KUKA KRL program: MyProgram_159().src

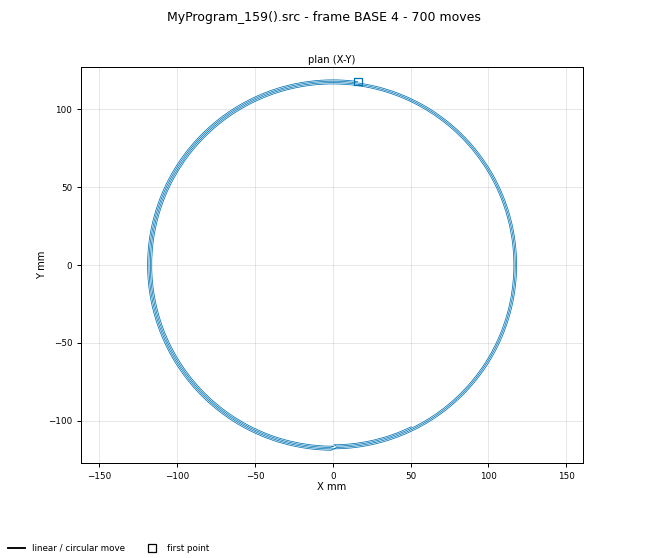
[picture p0: tool path of MyProgram_159().src in frame BASE 4, 700 of 700 moves have a stored position in this frame; points joined in program order, loops and branches not executed]
&ACCESS RVP
&REL 1
&PARAM TEMPLATE = C:\KRC\Roboter\Template\vorgabe
&PARAM EDITMASK = *
DEF MyProgram_159()
; ---- Setting reference (Base) ----
$BASE = BASE_DATA[4]

; --------------------------
; ---- Setting tool (TCP) ----
$TOOL = TOOL_DATA[3]
; --------------------------

$VEL.CP = VEL_APROX_PRINT
Startdeposition()
$VEL.CP = VEL_PRINT
LIN {X 16.0086,Y 117.8693,Z 122,A 78.2901,B 24.9375,C -1.8274,E1 25.0208,E2 367.7031} C_DIS
LIN {X 13.1111,Y 118.2266,Z 122,A 79.7079,B 24.9374,C -1.8281,E1 25.0168,E2 366.2845} C_DIS
LIN {X 10.2057,Y 118.5128,Z 122,A 81.1015,B 24.9374,C -1.8277,E1 25.013,E2 364.8927} C_DIS
LIN {X 6.984,Y 118.7447,Z 122,A 82.7398,B 24.9371,C -1.8315,E1 25.0084,E2 363.2462} C_DIS
LIN {X 2.9192,Y 118.9156,Z 122,A 84.6175,B 24.9374,C -1.8276,E1 25.0032,E2 361.3781} C_DIS
LIN {X 0,Y 118.9514,Z 122,A 86.0242,B 24.9374,C -1.8274,E1 24.9992,E2 359.9721} C_DIS
LIN {X -3.3524,Y 118.9023,Z 122,A 87.6856,B 24.9373,C -1.8291,E1 24.9946,E2 358.3065} C_DIS
LIN {X -7.2942,Y 118.7275,Z 122,A 89.5422,B 24.9375,C -1.8264,E1 24.9894,E2 356.4558} C_DIS
LIN {X -10.2057,Y 118.5128,Z 122,A 90.9498,B 24.9375,C -1.8258,E1 24.9855,E2 355.0489} C_DIS
LIN {X -13.2482,Y 118.2106,Z 122,A 92.3641,B 24.9377,C -1.8224,E1 24.9816,E2 353.6418} C_DIS
LIN {X -16.0086,Y 117.8693,Z 122,A 93.766,B 24.9377,C -1.8244,E1 24.9777,E2 352.2344} C_DIS
LIN {X -19.1267,Y 117.4024,Z 122,A 95.1851,B 24.938,C -1.8189,E1 24.9738,E2 350.8269} C_DIS
LIN {X -22.2224,Y 116.8552,Z 122,A 96.604,B 24.9384,C -1.8135,E1 24.9699,E2 349.4193} C_DIS
LIN {X -24.7181,Y 116.3543,Z 122,A 97.9954,B 24.9379,C -1.8198,E1 24.9661,E2 348.0115} C_DIS
LIN {X -27.4847,Y 115.7326,Z 122,A 99.4967,B 24.9376,C -1.8245,E1 24.962,E2 346.497} C_DIS
LIN {X -31.7259,Y 114.6425,Z 122,A 101.5145,B 24.938,C -1.8183,E1 24.9566,E2 344.491} C_DIS
LIN {X -34.5298,Y 113.8294,Z 122,A 102.9241,B 24.9381,C -1.8169,E1 24.9528,E2 343.0823} C_DIS
LIN {X -37.3129,Y 112.9477,Z 122,A 104.3341,B 24.9382,C -1.8154,E1 24.949,E2 341.6734} C_DIS
LIN {X -40.0735,Y 111.998,Z 122,A 105.7441,B 24.9383,C -1.8137,E1 24.9453,E2 340.2645} C_DIS
LIN {X -42.81,Y 110.9808,Z 122,A 107.1543,B 24.9385,C -1.812,E1 24.9417,E2 338.8553} C_DIS
LIN {X -45.5207,Y 109.8968,Z 122,A 108.5648,B 24.9385,C -1.8102,E1 24.938,E2 337.4459} C_DIS
LIN {X -48.204,Y 108.7465,Z 122,A 110.0438,B 24.9385,C -1.8113,E1 24.9342,E2 335.9608} C_DIS
LIN {X -50.8583,Y 107.5308,Z 122,A 111.3866,B 24.9388,C -1.8064,E1 24.9308,E2 334.6265} C_DIS
LIN {X -53.4819,Y 106.2503,Z 122,A 112.7979,B 24.939,C -1.8043,E1 24.9273,E2 333.2164} C_DIS
LIN {X -56.3435,Y 104.7592,Z 122,A 114.2234,B 24.9395,C -1.7961,E1 24.9238,E2 331.8064} C_DIS
LIN {X -58.6309,Y 103.4981,Z 122,A 115.6207,B 24.9393,C -1.7999,E1 24.9204,E2 330.396} C_DIS
LIN {X -61.1532,Y 102.028,Z 122,A 117.0324,B 24.9394,C -1.7976,E1 24.917,E2 328.9856} C_DIS
LIN {X -63.6387,Y 100.4965,Z 122,A 118.4444,B 24.9396,C -1.7952,E1 24.9137,E2 327.5749} C_DIS
LIN {X -66.0859,Y 98.9045,Z 122,A 119.8565,B 24.9398,C -1.7927,E1 24.9104,E2 326.1641} C_DIS
LIN {X -68.6207,Y 97.1619,Z 122,A 121.276,B 24.9401,C -1.787,E1 24.9071,E2 324.7532} C_DIS
LIN {X -70.8593,Y 95.5427,Z 122,A 122.6815,B 24.9401,C -1.7874,E1 24.9039,E2 323.3417} C_DIS
LIN {X -73.1827,Y 93.7749,Z 122,A 124.1704,B 24.9401,C -1.788,E1 24.9006,E2 321.8462} C_DIS
LIN {X -75.9227,Y 91.5678,Z 122,A 125.7971,B 24.9405,C -1.7813,E1 24.8971,E2 320.2291} C_DIS
LIN {X -78.7953,Y 89.1108,Z 122,A 127.6267,B 24.9408,C -1.7775,E1 24.8933,E2 318.4014} C_DIS
LIN {X -80.9584,Y 87.1502,Z 122,A 129.0403,B 24.941,C -1.7745,E1 24.8904,E2 316.9892} C_DIS
LIN {X -83.0728,Y 85.1372,Z 122,A 130.4536,B 24.9412,C -1.7715,E1 24.8875,E2 315.5773} C_DIS
LIN {X -85.1372,Y 83.0728,Z 122,A 131.8674,B 24.9414,C -1.7683,E1 24.8848,E2 314.165} C_DIS
LIN {X -87.2091,Y 80.8943,Z 122,A 133.2852,B 24.9417,C -1.7634,E1 24.8821,E2 312.7527} C_DIS
LIN {X -89.1108,Y 78.7953,Z 122,A 134.6952,B 24.9418,C -1.7618,E1 24.8794,E2 311.3402} C_DIS
LIN {X -91.2779,Y 76.2716,Z 122,A 136.1286,B 24.9426,C -1.7505,E1 24.8769,E2 309.9272} C_DIS
LIN {X -92.8698,Y 74.3279,Z 122,A 137.5238,B 24.9423,C -1.7551,E1 24.8744,E2 308.5145} C_DIS
LIN {X -94.6659,Y 72.0264,Z 122,A 138.9381,B 24.9425,C -1.7517,E1 24.872,E2 307.1016} C_DIS
LIN {X -96.405,Y 69.6815,Z 122,A 140.3529,B 24.9427,C -1.7482,E1 24.8697,E2 305.6883} C_DIS
LIN {X -98.0861,Y 67.2946,Z 122,A 141.7675,B 24.943,C -1.7446,E1 24.8674,E2 304.2753} C_DIS
LIN {X -99.708,Y 64.8672,Z 122,A 143.25,B 24.943,C -1.7438,E1 24.8651,E2 302.7872} C_DIS
LIN {X -101.2699,Y 62.4007,Z 122,A 144.5972,B 24.9434,C -1.7373,E1 24.8632,E2 301.4486} C_DIS
LIN {X -102.7708,Y 59.8966,Z 122,A 146.0608,B 24.9435,C -1.7356,E1 24.8611,E2 299.9814} C_DIS
LIN {X -104.2098,Y 57.3564,Z 122,A 147.4273,B 24.9439,C -1.7298,E1 24.8592,E2 298.6216} C_DIS
LIN {X -105.586,Y 54.7817,Z 122,A 148.8428,B 24.9442,C -1.726,E1 24.8574,E2 297.2076} C_DIS
LIN {X -106.8986,Y 52.174,Z 122,A 150.258,B 24.9444,C -1.7222,E1 24.8556,E2 295.794} C_DIS
LIN {X -108.1468,Y 49.5349,Z 122,A 151.6736,B 24.9447,C -1.7183,E1 24.854,E2 294.3799} C_DIS
LIN {X -109.3299,Y 46.8659,Z 122,A 153.0891,B 24.9449,C -1.7144,E1 24.8524,E2 292.9659} C_DIS
LIN {X -110.4471,Y 44.1687,Z 122,A 154.5047,B 24.9452,C -1.7104,E1 24.8509,E2 291.5519} C_DIS
LIN {X -111.4978,Y 41.4449,Z 122,A 155.9204,B 24.9454,C -1.7064,E1 24.8495,E2 290.1377} C_DIS
LIN {X -112.4813,Y 38.6961,Z 122,A 157.4741,B 24.9454,C -1.7082,E1 24.8481,E2 288.5709} C_DIS
LIN {X -113.588,Y 35.3084,Z 122,A 158.9656,B 24.9463,C -1.6934,E1 24.8468,E2 287.1063} C_DIS
LIN {X -114.4079,Y 32.5539,Z 122,A 160.4567,B 24.9463,C -1.6934,E1 24.8457,E2 285.6064} C_DIS
LIN {X -115.1723,Y 29.7364,Z 122,A 161.8742,B 24.9465,C -1.6894,E1 24.8446,E2 284.1903} C_DIS
LIN {X -116.0611,Y 26.0624,Z 122,A 163.7079,B 24.9469,C -1.6841,E1 24.8435,E2 282.3586} C_DIS
LIN {X -116.6658,Y 23.2063,Z 122,A 165.2237,B 24.9469,C -1.6841,E1 24.8426,E2 280.8337} C_DIS
LIN {X -117.4409,Y 18.8964,Z 122,A 167.248,B 24.9475,C -1.6737,E1 24.8417,E2 278.8222} C_DIS
LIN {X -117.8693,Y 16.0086,Z 122,A 168.6643,B 24.9478,C -1.6696,E1 24.8411,E2 277.4074} C_DIS
LIN {X -118.2266,Y 13.1111,Z 122,A 170.2103,B 24.9477,C -1.6708,E1 24.8406,E2 275.849} C_DIS
LIN {X -118.5128,Y 10.2057,Z 122,A 171.4964,B 24.9483,C -1.6612,E1 24.8403,E2 274.5782} C_DIS
LIN {X -118.7486,Y 6.9139,Z 122,A 172.9304,B 24.949,C -1.6495,E1 24.84,E2 273.1635} C_DIS
LIN {X -118.8708,Y 4.3783,Z 122,A 174.3286,B 24.9488,C -1.6529,E1 24.8399,E2 271.7489} C_DIS
LIN {X -118.9424,Y 1.4597,Z 122,A 175.741,B 24.9491,C -1.6485,E1 24.8398,E2 270.3382} C_DIS
LIN {X -118.9424,Y -1.4597,Z 122,A 177.3307,B 24.9489,C -1.6517,E1 24.8398,E2 268.7315} C_DIS
LIN {X -118.8081,Y -5.8367,Z 122,A 179.285,B 24.9497,C -1.6383,E1 24.84,E2 266.7973} C_DIS
LIN {X -118.6291,Y -8.7506,Z 122,A -179.2988,B 24.95,C -1.6342,E1 24.8403,E2 265.3825} C_DIS
LIN {X -118.3786,Y -11.6593,Z 122,A -177.7646,B 24.95,C -1.635,E1 24.8407,E2 263.837} C_DIS
LIN {X -118.0568,Y -14.5609,Z 122,A -176.2909,B 24.95,C -1.6334,E1 24.8412,E2 262.3584} C_DIS
LIN {X -117.6639,Y -17.4538,Z 122,A -175.0509,B 24.9507,C -1.6218,E1 24.8417,E2 261.1385} C_DIS
LIN {X -117.2002,Y -20.3362,Z 122,A -173.6352,B 24.951,C -1.6178,E1 24.8423,E2 259.724} C_DIS
LIN {X -116.6658,Y -23.2063,Z 122,A -172.2193,B 24.9512,C -1.6137,E1 24.8431,E2 258.3094} C_DIS
LIN {X -116.0611,Y -26.0624,Z 122,A -170.8033,B 24.9514,C -1.6097,E1 24.8439,E2 256.8947} C_DIS
LIN {X -115.3866,Y -28.9028,Z 122,A -169.3877,B 24.9517,C -1.6058,E1 24.8449,E2 255.4803} C_DIS
LIN {X -114.4951,Y -32.2459,Z 122,A -167.9472,B 24.9526,C -1.5911,E1 24.8459,E2 254.0663} C_DIS
LIN {X -113.8294,Y -34.5298,Z 122,A -166.5567,B 24.9522,C -1.5979,E1 24.847,E2 252.6516} C_DIS
LIN {X -112.9477,Y -37.3129,Z 122,A -165.1412,B 24.9524,C -1.594,E1 24.8482,E2 251.2372} C_DIS
LIN {X -111.9561,Y -40.1883,Z 122,A -163.7202,B 24.9528,C -1.5878,E1 24.8495,E2 249.8231} C_DIS
LIN {X -110.9808,Y -42.81,Z 122,A -162.3107,B 24.9528,C -1.5864,E1 24.8509,E2 248.4089} C_DIS
LIN {X -109.8968,Y -45.5207,Z 122,A -160.8955,B 24.9531,C -1.5826,E1 24.8524,E2 246.9948} C_DIS
LIN {X -108.7465,Y -48.204,Z 122,A -159.4806,B 24.9533,C -1.5789,E1 24.854,E2 245.5808} C_DIS
LIN {X -107.5308,Y -50.8583,Z 122,A -158.0655,B 24.9535,C -1.5753,E1 24.8557,E2 244.1668} C_DIS
LIN {X -106.0721,Y -53.8304,Z 122,A -156.6322,B 24.9542,C -1.5639,E1 24.8574,E2 242.7527} C_DIS
LIN {X -104.9058,Y -56.0733,Z 122,A -155.236,B 24.9539,C -1.5681,E1 24.8593,E2 241.3392} C_DIS
LIN {X -103.4981,Y -58.6309,Z 122,A -153.8215,B 24.9541,C -1.5646,E1 24.8612,E2 239.9255} C_DIS
LIN {X -102.028,Y -61.1532,Z 122,A -152.4071,B 24.9543,C -1.5612,E1 24.8632,E2 238.5121} C_DIS
LIN {X -100.4965,Y -63.6387,Z 122,A -150.9929,B 24.9545,C -1.5578,E1 24.8653,E2 237.0987} C_DIS
LIN {X -98.9045,Y -66.0859,Z 122,A -149.5789,B 24.9547,C -1.5545,E1 24.8675,E2 235.6854} C_DIS
LIN {X -97.2529,Y -68.4932,Z 122,A -148.1649,B 24.9549,C -1.5513,E1 24.8697,E2 234.2722} C_DIS
LIN {X -95.5427,Y -70.8593,Z 122,A -146.7512,B 24.9551,C -1.5481,E1 24.8721,E2 232.8592} C_DIS
LIN {X -93.7749,Y -73.1827,Z 122,A -145.3375,B 24.9553,C -1.545,E1 24.8745,E2 231.4463} C_DIS
LIN {X -91.9507,Y -75.462,Z 122,A -143.9239,B 24.9555,C -1.5419,E1 24.877,E2 230.0333} C_DIS
LIN {X -90.0711,Y -77.6958,Z 122,A -142.5105,B 24.9556,C -1.5389,E1 24.8795,E2 228.6206} C_DIS
LIN {X -88.1372,Y -79.8829,Z 122,A -141.0974,B 24.9558,C -1.536,E1 24.8822,E2 227.2081} C_DIS
LIN {X -86.1502,Y -82.0218,Z 122,A -139.6846,B 24.956,C -1.5332,E1 24.8849,E2 225.7959} C_DIS
LIN {X -84.1113,Y -84.1113,Z 122,A -138.2717,B 24.9561,C -1.5305,E1 24.8876,E2 224.3834} C_DIS
LIN {X -82.0218,Y -86.1502,Z 122,A -136.8593,B 24.9563,C -1.5278,E1 24.8905,E2 222.9716} C_DIS
LIN {X -79.8829,Y -88.1372,Z 122,A -135.4465,B 24.9564,C -1.5252,E1 24.8934,E2 221.5593} C_DIS
LIN {X -77.6958,Y -90.0711,Z 122,A -134.0346,B 24.9566,C -1.5227,E1 24.8963,E2 220.1478} C_DIS
LIN {X -75.462,Y -91.9507,Z 122,A -132.6226,B 24.9567,C -1.5202,E1 24.8994,E2 218.7362} C_DIS
LIN {X -72.8436,Y -94.0362,Z 122,A -131.1909,B 24.9573,C -1.5094,E1 24.9025,E2 217.325} C_DIS
LIN {X -70.8593,Y -95.5427,Z 122,A -129.7991,B 24.957,C -1.5156,E1 24.9056,E2 215.9134} C_DIS
LIN {X -68.4932,Y -97.2529,Z 122,A -128.3878,B 24.957,C -1.5135,E1 24.9088,E2 214.5024} C_DIS
LIN {X -66.0859,Y -98.9045,Z 122,A -126.9767,B 24.9572,C -1.5114,E1 24.9121,E2 213.0914} C_DIS
LIN {X -63.6387,Y -100.4965,Z 122,A -125.5655,B 24.9573,C -1.5094,E1 24.9154,E2 211.6805} C_DIS
LIN {X -61.1532,Y -102.028,Z 122,A -124.1547,B 24.9574,C -1.5075,E1 24.9188,E2 210.2699} C_DIS
LIN {X -58.6309,Y -103.4981,Z 122,A -122.7442,B 24.9575,C -1.5057,E1 24.9222,E2 208.8595} C_DIS
LIN {X -56.0733,Y -104.9058,Z 122,A -121.3338,B 24.9576,C -1.5039,E1 24.9257,E2 207.4491} C_DIS
LIN {X -53.4819,Y -106.2503,Z 122,A -119.886,B 24.9576,C -1.504,E1 24.9293,E2 205.9973} C_DIS
LIN {X -50.8583,Y -107.5308,Z 122,A -118.5141,B 24.9578,C -1.5008,E1 24.9327,E2 204.6295} C_DIS
LIN {X -48.204,Y -108.7465,Z 122,A -117.1043,B 24.9578,C -1.4994,E1 24.9363,E2 203.2197} C_DIS
LIN {X -45.5207,Y -109.8968,Z 122,A -115.695,B 24.958,C -1.498,E1 24.9399,E2 201.8104} C_DIS
LIN {X -42.81,Y -110.9808,Z 122,A -114.119,B 24.9576,C -1.5043,E1 24.9441,E2 200.2161} C_DIS
LIN {X -39.8038,Y -112.0926,Z 122,A -112.8631,B 24.9584,C -1.49,E1 24.9473,E2 198.9917} C_DIS
LIN {X -37.3129,Y -112.9477,Z 122,A -111.4682,B 24.9582,C -1.4946,E1 24.951,E2 197.5832} C_DIS
LIN {X -34.5298,Y -113.8294,Z 122,A -110.0595,B 24.9582,C -1.4936,E1 24.9548,E2 196.1743} C_DIS
LIN {X -31.6187,Y -114.6714,Z 122,A -108.6462,B 24.9584,C -1.4906,E1 24.9586,E2 194.7659} C_DIS
LIN {X -28.9028,Y -115.3866,Z 122,A -107.2432,B 24.9583,C -1.4921,E1 24.9624,E2 193.3575} C_DIS
LIN {X -26.0624,Y -116.0611,Z 122,A -105.8354,B 24.9583,C -1.4914,E1 24.9662,E2 191.9494} C_DIS
LIN {X -23.2063,Y -116.6658,Z 122,A -104.3529,B 24.9582,C -1.4943,E1 24.9703,E2 190.4583} C_DIS
LIN {X -19.7453,Y -117.2989,Z 122,A -102.732,B 24.9584,C -1.4904,E1 24.9747,E2 188.8451} C_DIS
LIN {X -16.0086,Y -117.8693,Z 122,A -100.8392,B 24.9582,C -1.4932,E1 24.98,E2 186.944} C_DIS
LIN {X -13.1111,Y -118.2266,Z 122,A -99.5036,B 24.9584,C -1.4898,E1 24.9837,E2 185.6156} C_DIS
LIN {X -10.2057,Y -118.5128,Z 122,A -98.0971,B 24.9584,C -1.4897,E1 24.9876,E2 184.2086} C_DIS
LIN {X -7.2942,Y -118.7275,Z 122,A -96.6908,B 24.9584,C -1.4897,E1 24.9915,E2 182.8017} C_DIS
LIN {X -4.3783,Y -118.8708,Z 122,A -95.2849,B 24.9584,C -1.4898,E1 24.9954,E2 181.3953} C_DIS
LIN {X -1.1166,Y -118.9445,Z 122,A -93.6416,B 24.9582,C -1.4934,E1 25,E2 179.7433} C_DIS
LIN {X -1.1166,Y -118.9445,Z 122,A -93.6416,B 24.9582,C -1.4934,E1 25,E2 179.7433} C_DIS
Enddeposition()
LIN {X 0.837,Y -118.0667,Z 122,A -93.3866,B 24.9591,C -1.4776,E1 25.0006,E2 179.5259} C_DIS
Startdeposition()
$VEL.CP = VEL_PRINT
LIN {X -2.5203,Y -118.0457,Z 122,A -95.0963,B 24.9593,C -1.4736,E1 24.9958,E2 181.2451} C_DIS
LIN {X -6.0284,Y -117.9191,Z 122,A -96.9279,B 24.9596,C -1.4677,E1 24.9907,E2 183.0911} C_DIS
LIN {X -9.7991,Y -117.6654,Z 122,A -98.7213,B 24.9596,C -1.4695,E1 24.9857,E2 184.8809} C_DIS
LIN {X -13.6232,Y -117.2835,Z 122,A -100.5453,B 24.9594,C -1.4716,E1 24.9806,E2 186.701} C_DIS
LIN {X -17.1647,Y -116.8191,Z 122,A -102.3364,B 24.9596,C -1.4694,E1 24.9757,E2 188.4989} C_DIS
LIN {X -20.8111,Y -116.2235,Z 122,A -104.0964,B 24.9594,C -1.4714,E1 24.9708,E2 190.2557} C_DIS
LIN {X -24.1501,Y -115.5766,Z 122,A -105.8865,B 24.9597,C -1.4659,E1 24.9659,E2 192.0609} C_DIS
LIN {X -28.319,Y -114.6262,Z 122,A -107.7431,B 24.9591,C -1.4767,E1 24.9609,E2 193.8945} C_DIS
LIN {X -31.6333,Y -113.7571,Z 122,A -109.4534,B 24.9592,C -1.4756,E1 24.9563,E2 195.61} C_DIS
LIN {X -35.4313,Y -112.6316,Z 122,A -111.4026,B 24.9592,C -1.4758,E1 24.9511,E2 197.562} C_DIS
LIN {X -39.6049,Y -111.2329,Z 122,A -113.4657,B 24.9589,C -1.4808,E1 24.9456,E2 199.6172} C_DIS
LIN {X -43.033,Y -109.9508,Z 122,A -115.3202,B 24.959,C -1.4791,E1 24.9408,E2 201.4797} C_DIS
LIN {X -46.5467,Y -108.5122,Z 122,A -117.2594,B 24.9591,C -1.4768,E1 24.9358,E2 203.4289} C_DIS
LIN {X -49.8822,Y -107.0176,Z 122,A -118.9207,B 24.9588,C -1.4837,E1 24.9316,E2 205.0777} C_DIS
LIN {X -52.9112,Y -105.5542,Z 122,A -120.5495,B 24.9586,C -1.4859,E1 24.9275,E2 206.7057} C_DIS
LIN {X -56.2696,Y -103.8014,Z 122,A -122.3858,B 24.9585,C -1.4884,E1 24.923,E2 208.541} C_DIS
LIN {X -59.4142,Y -102.0362,Z 122,A -125.1607,B 24.9608,C -1.4469,E1 24.9161,E2 211.4229} C_DIS
LIN {X -64.7113,Y -98.7602,Z 122,A -127.2367,B 24.9583,C -1.4921,E1 24.9114,E2 213.3982} C_DIS
LIN {X -67.4344,Y -96.9207,Z 122,A -128.7977,B 24.9581,C -1.4962,E1 24.9078,E2 214.9547} C_DIS
LIN {X -70.4261,Y -94.771,Z 122,A -130.6293,B 24.958,C -1.4974,E1 24.9037,E2 216.7899} C_DIS
LIN {X -73.6051,Y -92.3231,Z 122,A -133.3064,B 24.9595,C -1.47,E1 24.8977,E2 219.5422} C_DIS
LIN {X -77.5667,Y -89.0192,Z 122,A -134.7328,B 24.9567,C -1.5206,E1 24.8949,E2 220.8536} C_DIS
LIN {X -80.6537,Y -86.2328,Z 122,A -137.0863,B 24.9573,C -1.5103,E1 24.8899,E2 223.241} C_DIS
LIN {X -82.9849,Y -83.9912,Z 122,A -138.6859,B 24.9571,C -1.5124,E1 24.8867,E2 224.8424} C_DIS
LIN {X -85.3632,Y -81.5744,Z 122,A -140.3333,B 24.9569,C -1.5159,E1 24.8835,E2 226.4886} C_DIS
LIN {X -87.9813,Y -78.742,Z 122,A -142.2473,B 24.9569,C -1.5183,E1 24.8799,E2 228.4053} C_DIS
LIN {X -90.2888,Y -76.0878,Z 122,A -143.9596,B 24.9566,C -1.522,E1 24.8768,E2 230.1165} C_DIS
LIN {X -92.7396,Y -73.078,Z 122,A -145.7909,B 24.9562,C -1.5288,E1 24.8736,E2 231.9403} C_DIS
LIN {X -95.2869,Y -69.7238,Z 122,A -147.8273,B 24.9559,C -1.5342,E1 24.8702,E2 233.9737} C_DIS
LIN {X -97.3807,Y -66.7718,Z 122,A -149.545,B 24.9556,C -1.5402,E1 24.8675,E2 235.6854} C_DIS
LIN {X -99.1458,Y -64.1192,Z 122,A -151.191,B 24.9556,C -1.5401,E1 24.8649,E2 237.34} C_DIS
LIN {X -101.046,Y -61.0803,Z 122,A -152.8963,B 24.9552,C -1.5461,E1 24.8625,E2 239.0397} C_DIS
LIN {X -102.7863,Y -58.1065,Z 122,A -154.6916,B 24.9552,C -1.5455,E1 24.8599,E2 240.8458} C_DIS
LIN {X -104.6351,Y -54.7049,Z 122,A -156.4189,B 24.9546,C -1.557,E1 24.8577,E2 242.5548} C_DIS
LIN {X -106.1616,Y -51.6825,Z 122,A -158.3147,B 24.9549,C -1.5511,E1 24.8553,E2 244.4749} C_DIS
LIN {X -108.0733,Y -47.5535,Z 122,A -160.645,B 24.9549,C -1.5524,E1 24.8526,E2 246.8149} C_DIS
LIN {X -109.8468,Y -43.298,Z 122,A -162.6472,B 24.9539,C -1.5687,E1 24.8506,E2 248.7893} C_DIS
LIN {X -111.1689,Y -39.7858,Z 122,A -164.3767,B 24.9533,C -1.5779,E1 24.8489,E2 250.5067} C_DIS
LIN {X -112.2303,Y -36.681,Z 122,A -166.101,B 24.9533,C -1.5773,E1 24.8474,E2 252.2424} C_DIS
LIN {X -113.1981,Y -33.5739,Z 122,A -167.6026,B 24.9529,C -1.5853,E1 24.8462,E2 253.7335} C_DIS
LIN {X -114.0754,Y -30.4619,Z 122,A -169.6456,B 24.9538,C -1.5707,E1 24.8446,E2 255.8233} C_DIS
LIN {X -114.957,Y -26.9451,Z 122,A -170.7843,B 24.9519,C -1.6017,E1 24.8439,E2 256.8947} C_DIS
LIN {X -115.6853,Y -23.6207,Z 122,A -172.8482,B 24.9526,C -1.5899,E1 24.8427,E2 258.9989} C_DIS
LIN {X -116.6652,Y -18.173,Z 122,A -175.4722,B 24.952,C -1.601,E1 24.8415,E2 261.6121} C_DIS
LIN {X -117.2671,Y -13.7637,Z 122,A -177.5041,B 24.9512,C -1.6131,E1 24.8408,E2 263.6272} C_DIS
LIN {X -117.5907,Y -10.6525,Z 122,A -179.1069,B 24.9512,C -1.6145,E1 24.8403,E2 265.2362} C_DIS
LIN {X -117.8809,Y -6.7187,Z 122,A 178.9732,B 24.9508,C -1.6205,E1 24.84,E2 267.1535} C_DIS
LIN {X -118.0266,Y -3.2916,Z 122,A 177.31,B 24.9505,C -1.6259,E1 24.8398,E2 268.8137} C_DIS
LIN {X -118.0707,Y 0.6735,Z 122,A 175.2326,B 24.9505,C -1.6259,E1 24.8398,E2 270.9036} C_DIS
LIN {X -117.999,Y 4.191,Z 122,A 173.6973,B 24.9497,C -1.6385,E1 24.8399,E2 272.4182} C_DIS
LIN {X -117.8225,Y 7.6782,Z 122,A 172.1845,B 24.9489,C -1.6515,E1 24.8402,E2 273.9091} C_DIS
LIN {X -117.6304,Y 10.2227,Z 122,A 170.5906,B 24.9495,C -1.6409,E1 24.8405,E2 275.5378} C_DIS
LIN {X -117.2382,Y 14.0105,Z 122,A 168.906,B 24.9488,C -1.6537,E1 24.841,E2 277.2021} C_DIS
LIN {X -116.7982,Y 17.3099,Z 122,A 167.3023,B 24.9484,C -1.6594,E1 24.8417,E2 278.8018} C_DIS
LIN {X -116.0604,Y 21.7112,Z 122,A 163.9484,B 24.9509,C -1.6182,E1 24.8434,E2 282.2738} C_DIS
LIN {X -114.6541,Y 28.2045,Z 122,A 161.7774,B 24.9477,C -1.6712,E1 24.8447,E2 284.331} C_DIS
LIN {X -113.6608,Y 31.9732,Z 122,A 159.8393,B 24.9474,C -1.6753,E1 24.8462,E2 286.2706} C_DIS
LIN {X -112.4649,Y 35.9559,Z 122,A 157.7732,B 24.9471,C -1.6798,E1 24.8479,E2 288.3379} C_DIS
LIN {X -111.1922,Y 39.7203,Z 122,A 155.8664,B 24.9467,C -1.6867,E1 24.8496,E2 290.2391} C_DIS
LIN {X -109.9722,Y 42.9785,Z 122,A 154.2022,B 24.9463,C -1.693,E1 24.8513,E2 291.8977} C_DIS
LIN {X -108.4935,Y 46.5895,Z 122,A 152.254,B 24.9461,C -1.6965,E1 24.8534,E2 293.8483} C_DIS
LIN {X -106.9839,Y 49.9548,Z 122,A 150.543,B 24.9455,C -1.7052,E1 24.8553,E2 295.5479} C_DIS
LIN {X -105.5465,Y 52.9268,Z 122,A 148.9998,B 24.945,C -1.7125,E1 24.8572,E2 297.0821} C_DIS
LIN {X -104.1322,Y 55.6598,Z 122,A 147.2749,B 24.9454,C -1.7074,E1 24.8595,E2 298.8284} C_DIS
LIN {X -101.2999,Y 60.6614,Z 122,A 144.5478,B 24.9447,C -1.7181,E1 24.8633,E2 301.5441} C_DIS
LIN {X -99.4431,Y 63.6562,Z 122,A 142.8906,B 24.9442,C -1.7252,E1 24.8657,E2 303.1929} C_DIS
LIN {X -97.7178,Y 66.274,Z 122,A 141.3586,B 24.944,C -1.729,E1 24.8681,E2 304.7233} C_DIS
LIN {X -94.6762,Y 70.5522,Z 122,A 138.6995,B 24.9438,C -1.7314,E1 24.8725,E2 307.3897} C_DIS
LIN {X -92.2919,Y 73.6445,Z 122,A 136.8665,B 24.9433,C -1.739,E1 24.8756,E2 309.2131} C_DIS
LIN {X -89.7223,Y 76.7526,Z 122,A 134.9443,B 24.9429,C -1.7456,E1 24.8791,E2 311.1285} C_DIS
LIN {X -87.2765,Y 79.5236,Z 122,A 133.1183,B 24.9427,C -1.7489,E1 24.8825,E2 312.955} C_DIS
LIN {X -84.854,Y 82.1027,Z 122,A 131.4882,B 24.9422,C -1.7568,E1 24.8856,E2 314.5732} C_DIS
LIN {X -82.8543,Y 84.1202,Z 122,A 129.9947,B 24.9422,C -1.7553,E1 24.8885,E2 316.0766} C_DIS
LIN {X -79.8987,Y 86.9322,Z 122,A 127.9946,B 24.942,C -1.7592,E1 24.8926,E2 318.0757} C_DIS
LIN {X -77.3128,Y 89.241,Z 122,A 126.3016,B 24.9418,C -1.7626,E1 24.8962,E2 319.7672} C_DIS
LIN {X -74.5056,Y 91.5968,Z 122,A 124.5387,B 24.9415,C -1.7672,E1 24.8999,E2 321.5258} C_DIS
LIN {X -71.9353,Y 93.6288,Z 122,A 122.9307,B 24.9413,C -1.7699,E1 24.9035,E2 323.1334} C_DIS
LIN {X -69.1893,Y 95.6775,Z 122,A 121.105,B 24.9415,C -1.7665,E1 24.9076,E2 324.9736} C_DIS
LIN {X -66.0058,Y 97.8994,Z 122,A 119.3885,B 24.9408,C -1.7773,E1 24.9115,E2 326.6702} C_DIS
LIN {X -62.7591,Y 100.0118,Z 122,A 117.4417,B 24.9408,C -1.7781,E1 24.9161,E2 328.6213} C_DIS
LIN {X -59.6107,Y 101.9209,Z 122,A 115.4385,B 24.9411,C -1.7722,E1 24.921,E2 330.6446} C_DIS
LIN {X -55.9381,Y 103.9812,Z 122,A 113.5453,B 24.9405,C -1.7821,E1 24.9256,E2 332.5197} C_DIS
LIN {X -52.3168,Y 105.8489,Z 122,A 111.6507,B 24.94,C -1.7889,E1 24.9303,E2 334.4033} C_DIS
LIN {X -48.2993,Y 107.7415,Z 122,A 109.373,B 24.9401,C -1.787,E1 24.9361,E2 336.6911} C_DIS
LIN {X -44.3306,Y 109.4342,Z 122,A 107.3967,B 24.9396,C -1.795,E1 24.9411,E2 338.6528} C_DIS
LIN {X -41.4601,Y 110.5541,Z 122,A 105.9158,B 24.9394,C -1.7976,E1 24.945,E2 340.1306} C_DIS
LIN {X -36.9424,Y 112.1457,Z 122,A 103.6009,B 24.9392,C -1.8009,E1 24.9511,E2 342.4423} C_DIS
LIN {X -29.7282,Y 114.2688,Z 122,A 100.1226,B 24.9384,C -1.8123,E1 24.9604,E2 345.8992} C_DIS
LIN {X -24.7676,Y 115.4458,Z 122,A 97.7042,B 24.9381,C -1.817,E1 24.9669,E2 348.3096} C_DIS
LIN {X -20.6632,Y 116.2502,Z 122,A 95.4767,B 24.9386,C -1.81,E1 24.9731,E2 350.5561} C_DIS
LIN {X -17.9053,Y 116.7066,Z 122,A 94.0358,B 24.9388,C -1.8073,E1 24.9771,E2 352.0048} C_DIS
LIN {X -13.5104,Y 117.2967,Z 122,A 91.9668,B 24.9384,C -1.8122,E1 24.9828,E2 354.0636} C_DIS
LIN {X -10.5439,Y 117.6007,Z 122,A 90.4331,B 24.9387,C -1.8091,E1 24.987,E2 355.6054} C_DIS
LIN {X -6.7024,Y 117.8818,Z 122,A 88.5253,B 24.9387,C -1.8082,E1 24.9924,E2 357.5161} C_DIS
LIN {X -2.8061,Y 118.0404,Z 122,A 86.5758,B 24.9388,C -1.8063,E1 24.9978,E2 359.4706} C_DIS
LIN {X 0.8128,Y 118.0693,Z 122,A 84.9643,B 24.9384,C -1.813,E1 25.0023,E2 361.066} C_DIS
LIN {X 3.9593,Y 118.0061,Z 122,A 83.3553,B 24.9386,C -1.8095,E1 25.0068,E2 362.6828} C_DIS
LIN {X 7.629,Y 117.8258,Z 122,A 81.5262,B 24.9388,C -1.8075,E1 25.0119,E2 364.5161} C_DIS
LIN {X 11.4888,Y 117.5135,Z 122,A 79.5656,B 24.939,C -1.8037,E1 25.0174,E2 366.4846} C_DIS
LIN {X 15.0973,Y 117.1029,Z 122,A 77.9567,B 24.9386,C -1.8102,E1 25.0218,E2 368.0768} C_DIS
LIN {X 18.7081,Y 116.5823,Z 122,A 76.2518,B 24.9384,C -1.8126,E1 25.0265,E2 369.7746} C_DIS
LIN {X 21.6376,Y 116.0741,Z 122,A 74.618,B 24.939,C -1.8035,E1 25.031,E2 371.4281} C_DIS
LIN {X 25.4384,Y 115.2995,Z 122,A 72.9032,B 24.9386,C -1.8101,E1 25.0357,E2 373.125} C_DIS
LIN {X 28.7086,Y 114.5305,Z 122,A 71.2433,B 24.9387,C -1.8078,E1 25.0402,E2 374.788} C_DIS
LIN {X 32.2197,Y 113.5909,Z 122,A 69.4374,B 24.939,C -1.8047,E1 25.0451,E2 376.5982} C_DIS
LIN {X 36.8632,Y 112.1713,Z 122,A 67.1868,B 24.9388,C -1.8076,E1 25.051,E2 378.8378} C_DIS
LIN {X 40.1478,Y 111.0373,Z 122,A 65.3795,B 24.9392,C -1.8007,E1 25.0558,E2 380.658} C_DIS
LIN {X 43.7256,Y 109.6788,Z 122,A 63.5126,B 24.9394,C -1.7983,E1 25.0607,E2 382.5262} C_DIS
LIN {X 47.3382,Y 108.1672,Z 122,A 61.6992,B 24.9393,C -1.8002,E1 25.0653,E2 384.3309} C_DIS
LIN {X 50.8639,Y 106.555,Z 122,A 59.8248,B 24.9393,C -1.7983,E1 25.0701,E2 386.2051} C_DIS
LIN {X 54.2635,Y 104.8658,Z 122,A 58.0326,B 24.9393,C -1.7982,E1 25.0745,E2 387.9926} C_DIS
LIN {X 58.794,Y 102.3928,Z 122,A 55.0683,B 24.941,C -1.7736,E1 25.0819,E2 391.0063} C_DIS
LIN {X 61.9751,Y 100.5015,Z 122,A 53.7614,B 24.9397,C -1.7933,E1 25.0849,E2 392.2627} C_DIS
LIN {X 65.422,Y 98.2916,Z 122,A 51.754,B 24.94,C -1.7891,E1 25.0896,E2 394.2732} C_DIS
LIN {X 69.3897,Y 95.5316,Z 122,A 49.3063,B 24.9406,C -1.7804,E1 25.0952,E2 396.7332} C_DIS
LIN {X 74.6817,Y 91.4541,Z 122,A 46.2282,B 24.9405,C -1.782,E1 25.1019,E2 399.7961} C_DIS
LIN {X 76.9828,Y 89.5262,Z 122,A 44.6559,B 24.941,C -1.7737,E1 25.1053,E2 401.3818} C_DIS
LIN {X 79.5975,Y 87.2087,Z 122,A 42.9979,B 24.9411,C -1.7721,E1 25.1087,E2 403.0371} C_DIS
LIN {X 82.1318,Y 84.826,Z 122,A 41.3127,B 24.9414,C -1.7686,E1 25.1121,E2 404.7235} C_DIS
LIN {X 84.9177,Y 82.0366,Z 122,A 39.298,B 24.942,C -1.7597,E1 25.1161,E2 406.7505} C_DIS
LIN {X 87.8236,Y 78.9181,Z 122,A 37.3369,B 24.942,C -1.7601,E1 25.1198,E2 408.7022} C_DIS
LIN {X 90.2792,Y 76.099,Z 122,A 35.4408,B 24.9425,C -1.7519,E1 25.1232,E2 410.6089} C_DIS
LIN {X 92.7641,Y 73.0471,Z 122,A 33.3735,B 24.9433,C -1.7399,E1 25.1269,E2 412.6948} C_DIS
LIN {X 95.8142,Y 68.9994,Z 122,A 30.389,B 24.9453,C -1.7092,E1 25.1319,E2 415.7374} C_DIS
LIN {X 98.9075,Y 64.4878,Z 122,A 28.6197,B 24.943,C -1.7438,E1 25.1345,E2 417.4163} C_DIS
LIN {X 100.7914,Y 61.4991,Z 122,A 26.829,B 24.9435,C -1.7357,E1 25.1371,E2 419.2172} C_DIS
LIN {X 102.6551,Y 58.3374,Z 122,A 24.9447,B 24.9442,C -1.7259,E1 25.1398,E2 421.1147} C_DIS
LIN {X 104.2815,Y 55.3763,Z 122,A 22.6676,B 24.9464,C -1.6913,E1 25.1429,E2 423.4615} C_DIS
LIN {X 106.7024,Y 50.5572,Z 122,A 20.9929,B 24.944,C -1.7284,E1 25.1448,E2 425.0398} C_DIS
LIN {X 108.3694,Y 46.8743,Z 122,A 18.9427,B 24.9447,C -1.7185,E1 25.1471,E2 427.1021} C_DIS
LIN {X 109.7729,Y 43.4859,Z 122,A 17.1076,B 24.9452,C -1.7106,E1 25.149,E2 428.9457} C_DIS
LIN {X 110.9738,Y 40.3217,Z 122,A 15.5097,B 24.9453,C -1.7078,E1 25.1506,E2 430.5412} C_DIS
LIN {X 112.4838,Y 35.8975,Z 122,A 13.1867,B 24.9459,C -1.6983,E1 25.1527,E2 432.8735} C_DIS
LIN {X 113.5699,Y 32.294,Z 122,A 11.1941,B 24.9468,C -1.6848,E1 25.1542,E2 434.8866} C_DIS
LIN {X 114.7026,Y 28.0058,Z 122,A 9.2985,B 24.9465,C -1.6904,E1 25.1555,E2 436.7581} C_DIS
LIN {X 115.3591,Y 25.1651,Z 122,A 7.8907,B 24.9467,C -1.6863,E1 25.1564,E2 438.1674} C_DIS
LIN {X 116.0458,Y 21.7872,Z 122,A 6.102,B 24.9474,C -1.6754,E1 25.1573,E2 439.9713} C_DIS
LIN {X 116.7307,Y 17.7495,Z 122,A 4.2857,B 24.9473,C -1.6773,E1 25.1581,E2 441.7725} C_DIS
LIN {X 117.2253,Y 14.1206,Z 122,A 2.4448,B 24.9478,C -1.6685,E1 25.1588,E2 443.6231} C_DIS
LIN {X 117.6095,Y 10.4489,Z 122,A 0.6165,B 24.9483,C -1.6609,E1 25.1593,E2 445.4584} C_DIS
LIN {X 117.9009,Y 6.3574,Z 122,A -1.2194,B 24.9483,C -1.6619,E1 25.1596,E2 447.2811} C_DIS
LIN {X 118.0431,Y 2.6604,Z 122,A -3.1276,B 24.9489,C -1.6506,E1 25.1598,E2 449.2046} C_DIS
LIN {X 118.0662,Y -1.3229,Z 122,A -4.9914,B 24.9491,C -1.6477,E1 25.1598,E2 451.0644} C_DIS
LIN {X 117.9707,Y -4.8933,Z 122,A -6.7342,B 24.9495,C -1.6416,E1 25.1596,E2 452.8111} C_DIS
LIN {X 117.7525,Y -8.7089,Z 122,A -8.6255,B 24.95,C -1.6337,E1 25.1592,E2 454.7098} C_DIS
LIN {X 117.403,Y -12.5543,Z 122,A -10.4122,B 24.9501,C -1.6318,E1 25.1588,E2 456.4904} C_DIS
LIN {X 116.7698,Y -17.4967,Z 122,A -12.8436,B 24.9506,C -1.6232,E1 25.1578,E2 458.9276} C_DIS
LIN {X 116.1758,Y -21.0765,Z 122,A -14.4605,B 24.9506,C -1.6245,E1 25.1571,E2 460.5321} C_DIS
LIN {X 115.5186,Y -24.4307,Z 122,A -16.2942,B 24.9514,C -1.6106,E1 25.156,E2 462.3878} C_DIS
LIN {X 114.694,Y -28.041,Z 122,A -17.9805,B 24.9514,C -1.6102,E1 25.155,E2 464.0653} C_DIS
LIN {X 113.561,Y -32.3253,Z 122,A -20.0062,B 24.9514,C -1.6093,E1 25.1535,E2 466.0815} C_DIS
LIN {X 112.7649,Y -35.0012,Z 122,A -21.4172,B 24.9519,C -1.6023,E1 25.1523,E2 467.501} C_DIS
LIN {X 111.7466,Y -38.1298,Z 122,A -23.0616,B 24.9523,C -1.5949,E1 25.1509,E2 469.1536} C_DIS
LIN {X 109.8018,Y -43.4124,Z 122,A -25.6618,B 24.9525,C -1.5926,E1 25.1483,E2 471.7445} C_DIS
LIN {X 108.8078,Y -45.8462,Z 122,A -27.0053,B 24.9529,C -1.5854,E1 25.1469,E2 473.0976} C_DIS
LIN {X 107.3971,Y -49.0637,Z 122,A -29.0884,B 24.9543,C -1.562,E1 25.1444,E2 475.2246} C_DIS
LIN {X 105.9481,Y -52.1165,Z 122,A -30.2225,B 24.9531,C -1.5813,E1 25.1431,E2 476.3071} C_DIS
LIN {X 104.4755,Y -55.008,Z 122,A -31.8803,B 24.9537,C -1.5726,E1 25.141,E2 477.9767} C_DIS
LIN {X 102.6777,Y -58.2981,Z 122,A -34.2159,B 24.9554,C -1.5425,E1 25.1377,E2 480.3711} C_DIS
LIN {X 100.6521,Y -61.7282,Z 122,A -35.5684,B 24.9541,C -1.5646,E1 25.1358,E2 481.6645} C_DIS
LIN {X 99.2659,Y -63.9321,Z 122,A -36.8626,B 24.9544,C -1.5595,E1 25.1339,E2 482.9642} C_DIS
LIN {X 97.4119,Y -66.7256,Z 122,A -38.5749,B 24.9549,C -1.5508,E1 25.1312,E2 484.6886} C_DIS
LIN {X 95.3208,Y -69.6775,Z 122,A -40.222,B 24.9549,C -1.5511,E1 25.1285,E2 486.327} C_DIS
LIN {X 93.4104,Y -72.2188,Z 122,A -41.8012,B 24.9553,C -1.5452,E1 25.1258,E2 487.9127} C_DIS
LIN {X 90.888,Y -75.3684,Z 122,A -43.7419,B 24.9555,C -1.5407,E1 25.1224,E2 489.8549} C_DIS
LIN {X 88.769,Y -77.8532,Z 122,A -45.2922,B 24.9557,C -1.5382,E1 25.1196,E2 491.404} C_DIS
LIN {X 86.1907,Y -80.6984,Z 122,A -47.2295,B 24.9561,C -1.5299,E1 25.1159,E2 493.3524} C_DIS
LIN {X 83.5861,Y -83.395,Z 122,A -49.0444,B 24.9564,C -1.5256,E1 25.1123,E2 495.1698} C_DIS
LIN {X 80.8128,Y -86.0832,Z 122,A -50.7922,B 24.9564,C -1.5271,E1 25.1088,E2 496.9069} C_DIS
LIN {X 78.3666,Y -88.3174,Z 122,A -52.5432,B 24.9569,C -1.5165,E1 25.1052,E2 498.6759} C_DIS
LIN {X 75.4105,Y -90.853,Z 122,A -54.3221,B 24.9569,C -1.5175,E1 25.1014,E2 500.4456} C_DIS
LIN {X 72.9669,Y -92.8275,Z 122,A -55.9266,B 24.9573,C -1.5103,E1 25.0979,E2 502.061} C_DIS
LIN {X 69.8022,Y -95.2295,Z 122,A -57.8091,B 24.9573,C -1.5083,E1 25.0937,E2 503.9414} C_DIS
LIN {X 66.3591,Y -97.6602,Z 122,A -59.8285,B 24.9575,C -1.5053,E1 25.089,E2 505.9609} C_DIS
LIN {X 63.3384,Y -99.647,Z 122,A -61.5883,B 24.9578,C -1.5016,E1 25.0849,E2 507.7238} C_DIS
LIN {X 60.2444,Y -101.5463,Z 122,A -63.2975,B 24.9578,C -1.5008,E1 25.0808,E2 509.4296} C_DIS
LIN {X 57.431,Y -103.1635,Z 122,A -64.877,B 24.958,C -1.4977,E1 25.077,E2 511.0116} C_DIS
LIN {X 54.9132,Y -104.5254,Z 122,A -66.2932,B 24.9582,C -1.494,E1 25.0735,E2 512.4326} C_DIS
LIN {X 51.1791,Y -106.4035,Z 122,A -68.2784,B 24.9582,C -1.4927,E1 25.0685,E2 514.4156} C_DIS
LIN {X 48.365,Y -107.7119,Z 122,A -70.1066,B 24.9592,C -1.4754,E1 25.0638,E2 516.2802} C_DIS
LIN {X 45.2488,Y -109.0595,Z 122,A -71.3478,B 24.9583,C -1.4918,E1 25.0607,E2 517.4797} C_DIS
LIN {X 42.0392,Y -110.3348,Z 122,A -73.1085,B 24.9587,C -1.4855,E1 25.0561,E2 519.2513} C_DIS
LIN {X 37.8502,Y -111.8409,Z 122,A -75.2042,B 24.9587,C -1.4857,E1 25.0505,E2 521.3425} C_DIS
LIN {X 34.6866,Y -112.8625,Z 122,A -76.7917,B 24.9587,C -1.4849,E1 25.0463,E2 522.9288} C_DIS
LIN {X 31.7716,Y -113.7179,Z 122,A -78.2483,B 24.9587,C -1.4841,E1 25.0424,E2 524.385} C_DIS
LIN {X 28.4515,Y -114.5938,Z 122,A -80.1117,B 24.9593,C -1.4733,E1 25.0373,E2 526.2711} C_DIS
LIN {X 24.6659,Y -115.468,Z 122,A -81.9629,B 24.9593,C -1.4731,E1 25.0323,E2 528.1203} C_DIS
LIN {X 20.9564,Y -116.1974,Z 122,A -83.7084,B 24.9593,C -1.4756,E1 25.0275,E2 529.8577} C_DIS
LIN {X 17.2389,Y -116.8085,Z 122,A -85.5391,B 24.9593,C -1.4742,E1 25.0224,E2 531.6901} C_DIS
LIN {X 13.6552,Y -117.2798,Z 122,A -87.2476,B 24.9593,C -1.4751,E1 25.0177,E2 533.3949} C_DIS
LIN {X 10.7274,Y -117.5838,Z 122,A -88.6968,B 24.9593,C -1.4734,E1 25.0137,E2 534.8474} C_DIS
LIN {X 7.0363,Y -117.8633,Z 122,A -90.5836,B 24.9596,C -1.4685,E1 25.0084,E2 536.7451} C_DIS
LIN {X 3.2063,Y -118.0292,Z 122,A -92.3266,B 24.9593,C -1.4731,E1 25.0036,E2 538.4766} C_DIS
LIN {X 0.837,Y -118.0667,Z 122,A -93.3852,B 24.9591,C -1.477,E1 25.0006,E2 539.5259} C_DIS
Enddeposition()
LIN {X 0.837,Y -118.0667,Z 122,A -93.3852,B 24.9591,C -1.477,E1 25.0006,E2 539.5259} C_DIS
Startdeposition()
$VEL.CP = VEL_PRINT
LIN {X 2.2329,Y -117.1737,Z 122,A -92.0843,B 24.9567,C -1.5206,E1 25.0046,E2 538.1219} C_DIS
LIN {X 6.1534,Y -117.0337,Z 122,A -90.2165,B 24.9567,C -1.519,E1 25.0098,E2 536.2584} C_DIS
LIN {X 9.1687,Y -116.8359,Z 122,A -88.6968,B 24.9567,C -1.5216,E1 25.014,E2 534.7331} C_DIS
LIN {X 12.6784,Y -116.5081,Z 122,A -86.8958,B 24.9564,C -1.5262,E1 25.019,E2 532.9226} C_DIS
LIN {X 16.5077,Y -116.0265,Z 122,A -85.0735,B 24.9564,C -1.5245,E1 25.0241,E2 531.1058} C_DIS
LIN {X 20.2055,Y -115.4413,Z 122,A -83.2099,B 24.9563,C -1.5274,E1 25.0292,E2 529.2373} C_DIS
LIN {X 24.8306,Y -114.5344,Z 122,A -80.9907,B 24.9564,C -1.5255,E1 25.0353,E2 527.0253} C_DIS
LIN {X 31.0209,Y -113.0158,Z 122,A -77.7923,B 24.956,C -1.5324,E1 25.044,E2 523.8153} C_DIS
LIN {X 34.3709,Y -112.042,Z 122,A -76.2955,B 24.9564,C -1.5247,E1 25.0479,E2 522.3393} C_DIS
LIN {X 40.5699,Y -109.9496,Z 122,A -72.9334,B 24.9558,C -1.5364,E1 25.0568,E2 518.9563} C_DIS
LIN {X 44.0552,Y -108.5993,Z 122,A -71.1624,B 24.9558,C -1.5364,E1 25.0614,E2 517.1894} C_DIS
LIN {X 47.8128,Y -106.9987,Z 122,A -68.4477,B 24.9536,C -1.5732,E1 25.0686,E2 514.3941} C_DIS
LIN {X 52.2317,Y -104.9121,Z 122,A -66.7748,B 24.9554,C -1.5433,E1 25.0726,E2 512.7964} C_DIS
LIN {X 57.5055,Y -102.1173,Z 122,A -63.9084,B 24.9552,C -1.5459,E1 25.0796,E2 509.932} C_DIS
LIN {X 60.5941,Y -100.315,Z 122,A -62.2065,B 24.9552,C -1.547,E1 25.0837,E2 508.2328} C_DIS
LIN {X 63.038,Y -98.7976,Z 122,A -60.8136,B 24.955,C -1.5491,E1 25.087,E2 506.8394} C_DIS
LIN {X 65.7497,Y -97.0136,Z 122,A -59.1806,B 24.9547,C -1.5545,E1 25.0908,E2 505.1992} C_DIS
LIN {X 69.4003,Y -94.4367,Z 122,A -56.9666,B 24.9544,C -1.5604,E1 25.0958,E2 502.9789} C_DIS
LIN {X 72.5265,Y -92.0576,Z 122,A -55.0511,B 24.9541,C -1.5643,E1 25.1001,E2 501.0612} C_DIS
LIN {X 75.3489,Y -89.7638,Z 122,A -53.2085,B 24.9537,C -1.5714,E1 25.104,E2 499.2089} C_DIS
LIN {X 78.0611,Y -87.4136,Z 122,A -51.5338,B 24.9537,C -1.5717,E1 25.1075,E2 497.5401} C_DIS
LIN {X 80.8152,Y -84.8767,Z 122,A -49.6537,B 24.9533,C -1.5784,E1 25.1114,E2 495.6518} C_DIS
LIN {X 83.2316,Y -82.5057,Z 122,A -48.0614,B 24.9533,C -1.5795,E1 25.1145,E2 494.0636} C_DIS
LIN {X 85.6644,Y -79.9778,Z 122,A -46.279,B 24.9528,C -1.5871,E1 25.118,E2 492.2712} C_DIS
LIN {X 88.2538,Y -77.1098,Z 122,A -44.4813,B 24.9528,C -1.5876,E1 25.1213,E2 490.4803} C_DIS
LIN {X 90.788,Y -74.1104,Z 122,A -42.5318,B 24.9524,C -1.5941,E1 25.1248,E2 488.5244} C_DIS
LIN {X 93.1281,Y -71.1481,Z 122,A -40.6512,B 24.952,C -1.6008,E1 25.128,E2 486.6368} C_DIS
LIN {X 95.4616,Y -67.9834,Z 122,A -38.8192,B 24.952,C -1.6018,E1 25.131,E2 484.8114} C_DIS
LIN {X 97.5899,Y -64.8928,Z 122,A -36.9963,B 24.9516,C -1.6064,E1 25.1339,E2 482.9866} C_DIS
LIN {X 98.9936,Y -62.7326,Z 122,A -35.4857,B 24.9507,C -1.6222,E1 25.1362,E2 481.4465} C_DIS
LIN {X 101.7212,Y -58.2022,Z 122,A -32.5757,B 24.9493,C -1.6456,E1 25.1403,E2 478.4963} C_DIS
LIN {X 103.8897,Y -54.2381,Z 122,A -30.9325,B 24.9505,C -1.6247,E1 25.1424,E2 476.9111} C_DIS
LIN {X 106.8139,Y -48.2229,Z 122,A -27.7713,B 24.9503,C -1.6293,E1 25.1462,E2 473.756} C_DIS
LIN {X 108.1648,Y -45.1133,Z 122,A -26.0472,B 24.9497,C -1.6376,E1 25.148,E2 472.0217} C_DIS
LIN {X 109.1565,Y -42.6562,Z 122,A -24.2662,B 24.948,C -1.6653,E1 25.1499,E2 470.1852} C_DIS
LIN {X 110.6045,Y -38.7466,Z 122,A -22.1648,B 24.9474,C -1.6749,E1 25.1518,E2 468.0732} C_DIS
LIN {X 112.0245,Y -34.4273,Z 122,A -20.8552,B 24.9498,C -1.6375,E1 25.1529,E2 466.8591} C_DIS
LIN {X 113.6462,Y -28.627,Z 122,A -17.5926,B 24.9482,C -1.6622,E1 25.1553,E2 463.5569} C_DIS
LIN {X 114.8408,Y -23.3725,Z 122,A -14.973,B 24.9477,C -1.67,E1 25.1569,E2 460.9341} C_DIS
LIN {X 115.5836,Y -19.367,Z 122,A -13.1448,B 24.9478,C -1.6686,E1 25.1578,E2 459.1201} C_DIS
LIN {X 116.3434,Y -14.1098,Z 122,A -10.4102,B 24.9469,C -1.6837,E1 25.1588,E2 456.366} C_DIS
LIN {X 116.7227,Y -10.5131,Z 122,A -8.6653,B 24.9466,C -1.6884,E1 25.1593,E2 454.6204} C_DIS
LIN {X 117.0163,Y -6.4677,Z 122,A -6.7839,B 24.9465,C -1.6899,E1 25.1596,E2 452.7465} C_DIS
LIN {X 117.157,Y -3.0356,Z 122,A -5.0243,B 24.9459,C -1.6993,E1 25.1598,E2 450.9753} C_DIS
LIN {X 117.1929,Y 0.7665,Z 122,A -3.1979,B 24.9456,C -1.7038,E1 25.1598,E2 449.1492} C_DIS
LIN {X 117.0993,Y 4.7415,Z 122,A -1.2798,B 24.9453,C -1.7089,E1 25.1596,E2 447.2306} C_DIS
LIN {X 116.8996,Y 8.3249,Z 122,A 0.5213,B 24.9448,C -1.7168,E1 25.1593,E2 445.4214} C_DIS
LIN {X 116.5612,Y 12.1708,Z 122,A 2.3142,B 24.9447,C -1.7183,E1 25.1588,E2 443.6356} C_DIS
LIN {X 116.0992,Y 15.9963,Z 122,A 4.2208,B 24.9442,C -1.7255,E1 25.1581,E2 441.7234} C_DIS
LIN {X 115.661,Y 18.9041,Z 122,A 6.2142,B 24.9421,C -1.757,E1 25.1572,E2 439.6673} C_DIS
LIN {X 114.8604,Y 23.2773,Z 122,A 7.7701,B 24.9437,C -1.7339,E1 25.1564,E2 438.1749} C_DIS
LIN {X 114.1663,Y 26.4709,Z 122,A 9.3775,B 24.9433,C -1.7394,E1 25.1554,E2 436.5639} C_DIS
LIN {X 112.3088,Y 33.4876,Z 122,A 13.4248,B 24.941,C -1.7745,E1 25.1523,E2 432.4572} C_DIS
LIN {X 111.043,Y 37.4715,Z 122,A 14.8937,B 24.9424,C -1.7529,E1 25.1511,E2 431.0475} C_DIS
LIN {X 109.815,Y 40.9352,Z 122,A 16.7629,B 24.9418,C -1.7617,E1 25.1493,E2 429.168} C_DIS
LIN {X 108.4926,Y 44.3175,Z 122,A 18.468,B 24.9418,C -1.7636,E1 25.1475,E2 427.4679} C_DIS
LIN {X 107.0038,Y 47.8015,Z 122,A 20.4456,B 24.941,C -1.775,E1 25.1453,E2 425.4742} C_DIS
LIN {X 104.1698,Y 53.6975,Z 122,A 23.5738,B 24.9406,C -1.7806,E1 25.1414,E2 422.3493} C_DIS
LIN {X 102.3315,Y 57.1219,Z 122,A 25.3553,B 24.9406,C -1.7802,E1 25.139,E2 420.5781} C_DIS
LIN {X 100.584,Y 60.1488,Z 122,A 27.1439,B 24.94,C -1.7886,E1 25.1365,E2 418.7789} C_DIS
LIN {X 98.6949,Y 63.198,Z 122,A 28.6324,B 24.9406,C -1.7807,E1 25.1343,E2 417.3166} C_DIS
LIN {X 95.4234,Y 68.037,Z 122,A 31.7947,B 24.9391,C -1.8026,E1 25.1293,E2 414.1183} C_DIS
LIN {X 92.8954,Y 71.45,Z 122,A 33.9428,B 24.9385,C -1.8111,E1 25.1256,E2 411.9602} C_DIS
LIN {X 90.0761,Y 74.9731,Z 122,A 35.9191,B 24.9389,C -1.8055,E1 25.1222,E2 410.0064} C_DIS
LIN {X 87.5101,Y 77.9533,Z 122,A 37.8446,B 24.9386,C -1.8101,E1 25.1186,E2 408.0787} C_DIS
LIN {X 84.2577,Y 81.4575,Z 122,A 40.152,B 24.9383,C -1.8139,E1 25.1142,E2 405.7723} C_DIS
LIN {X 81.4721,Y 84.2436,Z 122,A 41.8353,B 24.9388,C -1.8066,E1 25.1109,E2 404.1133} C_DIS
LIN {X 79.559,Y 86.0536,Z 122,A 43.3974,B 24.9378,C -1.8222,E1 25.1077,E2 402.5209} C_DIS
LIN {X 76.9191,Y 88.4204,Z 122,A 45.0545,B 24.9378,C -1.8221,E1 25.1042,E2 400.8706} C_DIS
LIN {X 74.5696,Y 90.4114,Z 122,A 47.3904,B 24.9349,C -1.864,E1 25.099,E2 398.4446} C_DIS
LIN {X 70.3543,Y 93.7279,Z 122,A 49.2708,B 24.937,C -1.8339,E1 25.095,E2 396.6421} C_DIS
LIN {X 67.7783,Y 95.608,Z 122,A 50.9273,B 24.9365,C -1.8411,E1 25.0912,E2 394.9743} C_DIS
LIN {X 64.2522,Y 98.0122,Z 122,A 52.9051,B 24.9365,C -1.8395,E1 25.0866,E2 393.007} C_DIS
LIN {X 61.0346,Y 100.0473,Z 122,A 55.1652,B 24.9351,C -1.8609,E1 25.0811,E2 390.7034} C_DIS
LIN {X 57.6652,Y 102.0263,Z 122,A 56.8198,B 24.9357,C -1.8517,E1 25.0772,E2 389.0753} C_DIS
LIN {X 53.4416,Y 104.3008,Z 122,A 58.7076,B 24.937,C -1.8338,E1 25.0726,E2 387.2352} C_DIS
LIN {X 51.1247,Y 105.4565,Z 122,A 60.1806,B 24.9362,C -1.8449,E1 25.0689,E2 385.74} C_DIS
LIN {X 48.636,Y 106.6278,Z 122,A 61.6832,B 24.9356,C -1.8537,E1 25.065,E2 384.2203} C_DIS
LIN {X 44.4767,Y 108.4277,Z 122,A 63.7115,B 24.936,C -1.8476,E1 25.0599,E2 382.2113} C_DIS
LIN {X 41.48,Y 109.6087,Z 122,A 65.3213,B 24.9358,C -1.8507,E1 25.0557,E2 380.5976} C_DIS
LIN {X 37.9102,Y 110.895,Z 122,A 67.1907,B 24.9356,C -1.853,E1 25.0507,E2 378.7265} C_DIS
LIN {X 31.8086,Y 112.7958,Z 122,A 70.5869,B 24.9346,C -1.8677,E1 25.0416,E2 375.3015} C_DIS
LIN {X 26.9092,Y 114.0651,Z 122,A 72.7306,B 24.9356,C -1.8542,E1 25.0358,E2 373.193} C_DIS
LIN {X 24.1928,Y 114.6724,Z 122,A 74.3003,B 24.9349,C -1.8642,E1 25.0315,E2 371.6015} C_DIS
LIN {X 19.6272,Y 115.5401,Z 122,A 76.3642,B 24.9354,C -1.8558,E1 25.0259,E2 369.56} C_DIS
LIN {X 16.5196,Y 116.0248,Z 122,A 77.9175,B 24.9354,C -1.8569,E1 25.0216,E2 368.0053} C_DIS
LIN {X 12.7038,Y 116.5055,Z 122,A 79.6417,B 24.9358,C -1.8503,E1 25.0169,E2 366.2981} C_DIS
LIN {X 9.2628,Y 116.8283,Z 122,A 81.4783,B 24.9354,C -1.857,E1 25.0117,E2 364.4467} C_DIS
LIN {X 5.5023,Y 117.0666,Z 122,A 83.4092,B 24.9351,C -1.8609,E1 25.0063,E2 362.5072} C_DIS
LIN {X 1.599,Y 117.1854,Z 122,A 85.3104,B 24.9351,C -1.8603,E1 25.001,E2 360.6077} C_DIS
LIN {X -1.9022,Y 117.1798,Z 122,A 86.9671,B 24.9353,C -1.8575,E1 24.9964,E2 358.9577} C_DIS
LIN {X -5.5446,Y 117.0648,Z 122,A 88.8217,B 24.9351,C -1.8601,E1 24.9912,E2 357.0965} C_DIS
LIN {X -9.1806,Y 116.8349,Z 122,A 90.5178,B 24.9355,C -1.8556,E1 24.9865,E2 355.4104} C_DIS
LIN {X -12.8259,Y 116.4927,Z 122,A 92.1702,B 24.9359,C -1.8486,E1 24.982,E2 353.7737} C_DIS
LIN {X -17.7746,Y 115.8393,Z 122,A 94.6839,B 24.9359,C -1.8503,E1 24.975,E2 351.2541} C_DIS
LIN {X -20.8318,Y 115.3286,Z 122,A 96.281,B 24.9357,C -1.8527,E1 24.9706,E2 349.6497} C_DIS
LIN {X -24.056,Y 114.7005,Z 122,A 98.6748,B 24.9333,C -1.8859,E1 24.9638,E2 347.1741} C_DIS
LIN {X -29.1727,Y 113.506,Z 122,A 100.0749,B 24.9371,C -1.8323,E1 24.9604,E2 345.8993} C_DIS
LIN {X -31.3215,Y 112.9323,Z 122,A 102.237,B 24.9339,C -1.8779,E1 24.9543,E2 343.6255} C_DIS
LIN {X -35.943,Y 111.5472,Z 122,A 103.8881,B 24.9362,C -1.8443,E1 24.9501,E2 342.0512} C_DIS
LIN {X -39.1326,Y 110.4691,Z 122,A 105.6722,B 24.936,C -1.8482,E1 24.9453,E2 340.2545} C_DIS
LIN {X -42.9923,Y 109.0245,Z 122,A 107.5962,B 24.9364,C -1.8416,E1 24.9403,E2 338.3422} C_DIS
LIN {X -46.383,Y 107.6267,Z 122,A 109.5021,B 24.9363,C -1.8438,E1 24.9354,E2 336.4266} C_DIS
LIN {X -50.3034,Y 105.8512,Z 122,A 111.534,B 24.9367,C -1.8375,E1 24.9303,E2 334.4047} C_DIS
LIN {X -53.2426,Y 104.4025,Z 122,A 113.0653,B 24.9371,C -1.8319,E1 24.9265,E2 332.8828} C_DIS
LIN {X -56.1024,Y 102.8943,Z 122,A 114.6782,B 24.9371,C -1.8305,E1 24.9225,E2 331.2685} C_DIS
LIN {X -60.1212,Y 100.6003,Z 122,A 117.1652,B 24.9368,C -1.836,E1 24.9165,E2 328.761} C_DIS
LIN {X -63.8882,Y 98.2519,Z 122,A 119.2094,B 24.9375,C -1.8264,E1 24.9117,E2 326.733} C_DIS
LIN {X -66.249,Y 96.6755,Z 122,A 120.9737,B 24.9366,C -1.8397,E1 24.9075,E2 324.9311} C_DIS
LIN {X -69.1848,Y 94.5945,Z 122,A 122.4622,B 24.9376,C -1.8245,E1 24.9042,E2 323.4735} C_DIS
LIN {X -72.6113,Y 91.9905,Z 122,A 124.4052,B 24.9384,C -1.8132,E1 24.9,E2 321.5504} C_DIS
LIN {X -75.5161,Y 89.6236,Z 122,A 126.1541,B 24.9389,C -1.8056,E1 24.8963,E2 319.8129} C_DIS
LIN {X -78.363,Y 87.1433,Z 122,A 128.1921,B 24.9386,C -1.8094,E1 24.892,E2 317.7577} C_DIS
LIN {X -81.3301,Y 84.3805,Z 122,A 130.1049,B 24.9391,C -1.8018,E1 24.8881,E2 315.8552} C_DIS
LIN {X -84.1552,Y 81.5639,Z 122,A 132.0909,B 24.9394,C -1.7985,E1 24.8842,E2 313.8686} C_DIS
LIN {X -86.9967,Y 78.5268,Z 122,A 134.3485,B 24.9391,C -1.8028,E1 24.8799,E2 311.5909} C_DIS
LIN {X -89.9437,Y 75.1324,Z 122,A 136.293,B 24.9402,C -1.7864,E1 24.8764,E2 309.6764} C_DIS
LIN {X -91.9084,Y 72.7152,Z 122,A 137.7209,B 24.9407,C -1.7784,E1 24.874,E2 308.261} C_DIS
LIN {X -94.6867,Y 69.0589,Z 122,A 140.4066,B 24.9399,C -1.7907,E1 24.8694,E2 305.5331} C_DIS
LIN {X -98.4771,Y 63.5374,Z 122,A 143.3567,B 24.9414,C -1.7679,E1 24.8649,E2 302.6226} C_DIS
LIN {X -102.4781,Y 56.8593,Z 122,A 147.3456,B 24.9417,C -1.7644,E1 24.8592,E2 298.6214} C_DIS
LIN {X -104.3186,Y 53.4068,Z 122,A 149.1679,B 24.9423,C -1.7549,E1 24.8569,E2 296.8119} C_DIS
LIN {X -106.1195,Y 49.7333,Z 122,A 151.1632,B 24.9427,C -1.7486,E1 24.8545,E2 294.8208} C_DIS
LIN {X -107.5031,Y 46.6666,Z 122,A 152.8954,B 24.9427,C -1.7472,E1 24.8525,E2 293.0824} C_DIS
LIN {X -108.9637,Y 43.1471,Z 122,A 154.7053,B 24.9433,C -1.7393,E1 24.8506,E2 291.2815} C_DIS
LIN {X -110.3664,Y 39.425,Z 122,A 157.0121,B 24.9427,C -1.7482,E1 24.8484,E2 288.9403} C_DIS
LIN {X -111.4036,Y 36.3868,Z 122,A 158.265,B 24.9439,C -1.7301,E1 24.8473,E2 287.7233} C_DIS
LIN {X -112.4075,Y 33.1549,Z 122,A 159.9393,B 24.9442,C -1.7257,E1 24.846,E2 286.05} C_DIS
LIN {X -113.431,Y 29.4643,Z 122,A 161.7208,B 24.9448,C -1.7159,E1 24.8447,E2 284.2813} C_DIS
LIN {X -114.545,Y 24.7811,Z 122,A 164.2821,B 24.9448,C -1.7169,E1 24.8431,E2 281.7026} C_DIS
LIN {X -115.4799,Y 19.9872,Z 122,A 166.7415,B 24.9451,C -1.7121,E1 24.8418,E2 279.2401} C_DIS
LIN {X -115.9936,Y 16.7391,Z 122,A 168.3205,B 24.9455,C -1.7057,E1 24.8412,E2 277.667} C_DIS
LIN {X -116.5181,Y 12.5828,Z 122,A 170.2609,B 24.9462,C -1.6946,E1 24.8406,E2 275.7414} C_DIS
LIN {X -116.8758,Y 8.6693,Z 122,A 172.6405,B 24.9454,C -1.7073,E1 24.8401,E2 273.3173} C_DIS
LIN {X -117.0876,Y 5.0135,Z 122,A 173.9596,B 24.947,C -1.682,E1 24.8399,E2 272.0507} C_DIS
LIN {X -117.1912,Y -1.0187,Z 122,A 177.0142,B 24.9473,C -1.6766,E1 24.8399,E2 268.9903} C_DIS
LIN {X -117.1315,Y -3.8657,Z 122,A 178.8061,B 24.9466,C -1.6887,E1 24.8399,E2 267.1588} C_DIS
LIN {X -116.9482,Y -7.606,Z 122,A -179.3118,B 24.9468,C -1.6849,E1 24.8403,E2 265.2744} C_DIS
LIN {X -116.6229,Y -11.5815,Z 122,A -177.7346,B 24.9482,C -1.6631,E1 24.8407,E2 263.7399} C_DIS
LIN {X -116.2271,Y -15.0301,Z 122,A -175.4493,B 24.947,C -1.6822,E1 24.8416,E2 261.3952} C_DIS
LIN {X -115.5129,Y -19.7898,Z 122,A -173.7046,B 24.949,C -1.6493,E1 24.8423,E2 259.7186} C_DIS
LIN {X -114.3466,Y -25.6905,Z 122,A -170.6649,B 24.9493,C -1.6442,E1 24.8441,E2 256.6733} C_DIS
LIN {X -113.1276,Y -30.6071,Z 122,A -168.2752,B 24.95,C -1.6329,E1 24.8457,E2 254.2966} C_DIS
LIN {X -112.0109,Y -34.4715,Z 122,A -166.3427,B 24.9505,C -1.6255,E1 24.8473,E2 252.3706} C_DIS
LIN {X -111.1012,Y -37.2989,Z 122,A -164.7769,B 24.9505,C -1.6258,E1 24.8486,E2 250.795} C_DIS
LIN {X -109.7278,Y -41.1654,Z 122,A -162.7797,B 24.9509,C -1.6195,E1 24.8505,E2 248.8017} C_DIS
LIN {X -108.5596,Y -44.1528,Z 122,A -160.6906,B 24.9498,C -1.6367,E1 24.8528,E2 246.6597} C_DIS
LIN {X -106.8646,Y -48.1103,Z 122,A -159.4353,B 24.9523,C -1.595,E1 24.8541,E2 245.4971} C_DIS
LIN {X -105.3375,Y -51.3724,Z 122,A -157.2978,B 24.9517,C -1.6057,E1 24.8567,E2 243.3225} C_DIS
LIN {X -103.6584,Y -54.6771,Z 122,A -155.5363,B 24.9521,C -1.5985,E1 24.859,E2 241.5686} C_DIS
LIN {X -101.777,Y -58.1051,Z 122,A -153.5785,B 24.9523,C -1.5952,E1 24.8616,E2 239.6084} C_DIS
LIN {X -99.8405,Y -61.3749,Z 122,A -151.7438,B 24.9527,C -1.5893,E1 24.8643,E2 237.7785} C_DIS
LIN {X -97.5115,Y -65.0117,Z 122,A -149.3737,B 24.9523,C -1.5947,E1 24.868,E2 235.3835} C_DIS
LIN {X -94.6708,Y -69.0806,Z 122,A -147.4589,B 24.954,C -1.567,E1 24.871,E2 233.5254} C_DIS
LIN {X -91.7372,Y -72.9319,Z 122,A -144.7186,B 24.9534,C -1.577,E1 24.8757,E2 230.7483} C_DIS
LIN {X -89.5309,Y -75.6248,Z 122,A -142.5988,B 24.9526,C -1.5908,E1 24.8796,E2 228.5858} C_DIS
LIN {X -86.8517,Y -78.6887,Z 122,A -141.0136,B 24.9539,C -1.5689,E1 24.8825,E2 227.0457} C_DIS
LIN {X -84.3201,Y -81.3928,Z 122,A -139.3401,B 24.9545,C -1.5591,E1 24.8856,E2 225.3882} C_DIS
LIN {X -80.7372,Y -84.9502,Z 122,A -136.803,B 24.9545,C -1.5567,E1 24.8907,E2 222.8461} C_DIS
LIN {X -78.1543,Y -87.3302,Z 122,A -135.3011,B 24.9553,C -1.5441,E1 24.8938,E2 221.3683} C_DIS
LIN {X -75.0223,Y -90.0349,Z 122,A -132.5963,B 24.9538,C -1.5695,E1 24.8997,E2 218.5925} C_DIS
LIN {X -72.007,Y -92.4662,Z 122,A -131.0942,B 24.955,C -1.5491,E1 24.9029,E2 217.1336} C_DIS
LIN {X -69.4076,Y -94.4313,Z 122,A -129.5408,B 24.9553,C -1.5446,E1 24.9064,E2 215.5853} C_DIS
LIN {X -66.3755,Y -96.5885,Z 122,A -127.6069,B 24.9552,C -1.5465,E1 24.9108,E2 213.6403} C_DIS
LIN {X -63.8579,Y -98.2713,Z 122,A -125.8893,B 24.9547,C -1.5544,E1 24.9149,E2 211.8982} C_DIS
LIN {X -58.595,Y -101.4955,Z 122,A -123.242,B 24.9559,C -1.5338,E1 24.9211,E2 209.2918} C_DIS
LIN {X -55.844,Y -103.0345,Z 122,A -121.6409,B 24.9559,C -1.5343,E1 24.9251,E2 207.6849} C_DIS
LIN {X -52.3406,Y -104.8581,Z 122,A -119.9672,B 24.9567,C -1.5206,E1 24.9292,E2 206.0393} C_DIS
LIN {X -49.5294,Y -106.2144,Z 122,A -118.1769,B 24.9561,C -1.5304,E1 24.9337,E2 204.2213} C_DIS
LIN {X -45.8064,Y -107.8728,Z 122,A -116.1951,B 24.9563,C -1.5277,E1 24.9388,E2 202.2411} C_DIS
LIN {X -42.6733,Y -109.1498,Z 122,A -114.5445,B 24.9563,C -1.5259,E1 24.9431,E2 200.5912} C_DIS
LIN {X -38.5648,Y -110.6683,Z 122,A -111.9294,B 24.9553,C -1.5451,E1 24.9501,E2 197.9254} C_DIS
LIN {X -34.9152,Y -111.8733,Z 122,A -110.3115,B 24.956,C -1.532,E1 24.9543,E2 196.3357} C_DIS
LIN {X -30.7053,Y -113.1011,Z 122,A -108.3841,B 24.9567,C -1.5209,E1 24.9595,E2 194.4315} C_DIS
LIN {X -27.043,Y -114.0341,Z 122,A -105.987,B 24.9553,C -1.5445,E1 24.9661,E2 191.9751} C_DIS
LIN {X -23.0407,Y -114.909,Z 122,A -104.4647,B 24.9566,C -1.522,E1 24.9702,E2 190.5044} C_DIS
LIN {X -19.4686,Y -115.5666,Z 122,A -102.7373,B 24.9568,C -1.5193,E1 24.9749,E2 188.7817} C_DIS
LIN {X -15.9672,Y -116.1033,Z 122,A -100.9327,B 24.9566,C -1.5221,E1 24.9799,E2 186.9689} C_DIS
LIN {X -12.3989,Y -116.5374,Z 122,A -99.2642,B 24.9568,C -1.5179,E1 24.9845,E2 185.3094} C_DIS
LIN {X -9.0463,Y -116.8456,Z 122,A -97.5151,B 24.9566,C -1.5225,E1 24.9894,E2 183.5486} C_DIS
LIN {X -5.2359,Y -117.0781,Z 122,A -95.7181,B 24.9567,C -1.5195,E1 24.9944,E2 181.7583} C_DIS
LIN {X -1.5496,Y -117.1863,Z 122,A -93.8187,B 24.9565,C -1.5241,E1 24.9997,E2 179.8477} C_DIS
LIN {X -1.5496,Y -117.1863,Z 122,A -93.8187,B 24.9565,C -1.5241,E1 24.9997,E2 179.8477} C_DIS
Enddeposition()
LIN {X 0.8152,Y -116.3142,Z 122,A -92.8741,B 24.9561,C -1.5301,E1 25.0024,E2 178.8891} C_DIS
Startdeposition()
$VEL.CP = VEL_PRINT
LIN {X -2.9207,Y -116.283,Z 122,A -95.5224,B 24.9582,C -1.4936,E1 24.9948,E2 181.6239} C_DIS
LIN {X -6.261,Y -116.1493,Z 122,A -97.0516,B 24.9579,C -1.4987,E1 24.9905,E2 183.1414} C_DIS
LIN {X -10.0289,Y -115.8866,Z 122,A -98.9569,B 24.958,C -1.4967,E1 24.9852,E2 185.0522} C_DIS
LIN {X -13.4575,Y -115.5367,Z 122,A -100.5833,B 24.9578,C -1.5001,E1 24.9807,E2 186.6716} C_DIS
LIN {X -17.0677,Y -115.061,Z 122,A -102.5324,B 24.9582,C -1.4936,E1 24.9753,E2 188.6375} C_DIS
LIN {X -21.0059,Y -114.4061,Z 122,A -104.2204,B 24.9575,C -1.5065,E1 24.9707,E2 190.2967} C_DIS
LIN {X -27.5379,Y -113.0111,Z 122,A -107.6616,B 24.9578,C -1.5014,E1 24.9613,E2 193.7543} C_DIS
LIN {X -30.7866,Y -112.1706,Z 122,A -109.3709,B 24.9578,C -1.5,E1 24.9567,E2 195.4695} C_DIS
LIN {X -34.765,Y -111.0015,Z 122,A -111.6874,B 24.9584,C -1.4896,E1 24.9504,E2 197.8146} C_DIS
LIN {X -37.85,Y -109.9896,Z 122,A -113.0388,B 24.9578,C -1.5016,E1 24.9469,E2 199.14} C_DIS
LIN {X -40.8467,Y -108.9106,Z 122,A -114.5672,B 24.9576,C -1.5048,E1 24.9429,E2 200.664} C_DIS
LIN {X -44.335,Y -107.5384,Z 122,A -116.4028,B 24.9574,C -1.5071,E1 24.9382,E2 202.4982} C_DIS
LIN {X -47.6791,Y -106.0969,Z 122,A -118.1793,B 24.9573,C -1.5098,E1 24.9336,E2 204.2725} C_DIS
LIN {X -51.5787,Y -104.2568,Z 122,A -120.2761,B 24.9571,C -1.5136,E1 24.9283,E2 206.3658} C_DIS
LIN {X -54.8253,Y -102.5888,Z 122,A -122.1607,B 24.9571,C -1.5122,E1 24.9237,E2 208.2588} C_DIS
LIN {X -57.8284,Y -100.9244,Z 122,A -123.8171,B 24.9569,C -1.5161,E1 24.9196,E2 209.9109} C_DIS
LIN {X -63.1,Y -97.7155,Z 122,A -126.9855,B 24.9569,C -1.5152,E1 24.9121,E2 213.0912} C_DIS
LIN {X -66.5425,Y -95.4042,Z 122,A -128.9375,B 24.9566,C -1.5224,E1 24.9076,E2 215.0326} C_DIS
LIN {X -69.7083,Y -93.1162,Z 122,A -130.848,B 24.9564,C -1.5263,E1 24.9033,E2 216.9405} C_DIS
LIN {X -71.954,Y -91.392,Z 122,A -133.2068,B 24.9585,C -1.4887,E1 24.898,E2 219.3976} C_DIS
LIN {X -76.5367,Y -87.5898,Z 122,A -135.2399,B 24.956,C -1.5318,E1 24.8939,E2 221.3362} C_DIS
LIN {X -78.4312,Y -85.898,Z 122,A -137.239,B 24.9577,C -1.5033,E1 24.8896,E2 223.4111} C_DIS
LIN {X -82.2524,Y -82.2489,Z 122,A -139.1645,B 24.9558,C -1.5368,E1 24.8859,E2 225.2651} C_DIS
LIN {X -84.7769,Y -79.6412,Z 122,A -140.8811,B 24.9554,C -1.5437,E1 24.8826,E2 226.9725} C_DIS
LIN {X -88.2938,Y -75.7244,Z 122,A -143.5346,B 24.9552,C -1.5471,E1 24.8777,E2 229.6299} C_DIS
LIN {X -90.7136,Y -72.808,Z 122,A -145.8235,B 24.9559,C -1.5342,E1 24.8736,E2 231.9602} C_DIS
LIN {X -93.0406,Y -69.809,Z 122,A -147.1967,B 24.9544,C -1.5592,E1 24.8714,E2 233.2803} C_DIS
LIN {X -95.4988,Y -66.4064,Z 122,A -149.81,B 24.9554,C -1.5421,E1 24.8671,E2 235.9473} C_DIS
LIN {X -97.7123,Y -63.1051,Z 122,A -151.1935,B 24.9538,C -1.5707,E1 24.8651,E2 237.2696} C_DIS
LIN {X -99.3509,Y -60.4917,Z 122,A -152.7308,B 24.9536,C -1.574,E1 24.8628,E2 238.8069} C_DIS
LIN {X -100.7662,Y -58.1037,Z 122,A -154.2067,B 24.9536,C -1.5732,E1 24.8607,E2 240.2923} C_DIS
LIN {X -102.6455,Y -54.7182,Z 122,A -156.1368,B 24.9534,C -1.5775,E1 24.8581,E2 242.2224} C_DIS
LIN {X -104.2315,Y -51.6298,Z 122,A -157.7477,B 24.9528,C -1.5864,E1 24.8561,E2 243.8207} C_DIS
LIN {X -105.8671,Y -48.1892,Z 122,A -159.8181,B 24.953,C -1.5838,E1 24.8536,E2 245.9085} C_DIS
LIN {X -107.9851,Y -43.2376,Z 122,A -162.4722,B 24.9525,C -1.5915,E1 24.8508,E2 248.559} C_DIS
LIN {X -109.2218,Y -40.0058,Z 122,A -164.3294,B 24.9526,C -1.5904,E1 24.849,E2 250.4293} C_DIS
LIN {X -110.6867,Y -35.7531,Z 122,A -166.321,B 24.9517,C -1.6062,E1 24.8472,E2 252.3947} C_DIS
LIN {X -111.7712,Y -32.207,Z 122,A -168.2516,B 24.9516,C -1.6076,E1 24.8457,E2 254.3332} C_DIS
LIN {X -113.1327,Y -27.0391,Z 122,A -170.9038,B 24.9511,C -1.6149,E1 24.8439,E2 256.9834} C_DIS
LIN {X -114.4847,Y -20.5692,Z 122,A -175.0783,B 24.9527,C -1.5885,E1 24.8416,E2 261.2456} C_DIS
LIN {X -115.4106,Y -14.5059,Z 122,A -177.3656,B 24.9504,C -1.6274,E1 24.8408,E2 263.4538} C_DIS
LIN {X -116.0087,Y -8.4998,Z 122,A 178.9604,B 24.9515,C -1.6091,E1 24.84,E2 267.1936} C_DIS
LIN {X -116.2869,Y -2.75,Z 122,A 175.9407,B 24.9514,C -1.611,E1 24.8398,E2 270.2268} C_DIS
LIN {X -116.2594,Y 3.6888,Z 122,A 174.2619,B 24.947,C -1.681,E1 24.8398,E2 271.7488} C_DIS
LIN {X -115.896,Y 9.919,Z 122,A 170.6508,B 24.9478,C -1.6692,E1 24.8405,E2 275.4097} C_DIS
LIN {X -115.5565,Y 13.2886,Z 122,A 168.9497,B 24.9475,C -1.6734,E1 24.841,E2 277.1111} C_DIS
LIN {X -114.82,Y 18.6157,Z 122,A 166.2979,B 24.947,C -1.6819,E1 24.8421,E2 279.7585} C_DIS
LIN {X -114.1857,Y 22.1695,Z 122,A 164.5908,B 24.9464,C -1.6905,E1 24.843,E2 281.4551} C_DIS
LIN {X -112.8242,Y 28.3019,Z 122,A 161.361,B 24.9462,C -1.695,E1 24.845,E2 284.6932} C_DIS
LIN {X -111.7281,Y 32.3592,Z 122,A 159.3227,B 24.9457,C -1.7029,E1 24.8465,E2 286.7245} C_DIS
LIN {X -110.7462,Y 35.5693,Z 122,A 157.8573,B 24.9448,C -1.7157,E1 24.8477,E2 288.1677} C_DIS
LIN {X -108.7962,Y 41.1489,Z 122,A 154.8202,B 24.9446,C -1.7197,E1 24.8506,E2 291.2124} C_DIS
LIN {X -107.4894,Y 44.4554,Z 122,A 152.9523,B 24.9446,C -1.7204,E1 24.8525,E2 293.0892} C_DIS
LIN {X -106.1503,Y 47.5607,Z 122,A 151.0707,B 24.9448,C -1.7169,E1 24.8547,E2 294.9896} C_DIS
LIN {X -104.173,Y 51.7477,Z 122,A 149.0697,B 24.9436,C -1.735,E1 24.8571,E2 296.9581} C_DIS
LIN {X -102.3836,Y 55.2043,Z 122,A 147.1744,B 24.9432,C -1.7416,E1 24.8595,E2 298.8478} C_DIS
LIN {X -99.031,Y 61.018,Z 122,A 143.7106,B 24.9429,C -1.7448,E1 24.8644,E2 302.322} C_DIS
LIN {X -95.346,Y 66.6263,Z 122,A 140.5889,B 24.9418,C -1.7616,E1 24.8693,E2 305.4193} C_DIS
LIN {X -91.5469,Y 71.7581,Z 122,A 137.2926,B 24.9417,C -1.7639,E1 24.8748,E2 308.7258} C_DIS
LIN {X -89.5669,Y 74.2134,Z 122,A 135.148,B 24.943,C -1.7441,E1 24.8787,E2 310.9275} C_DIS
LIN {X -86.7157,Y 77.5257,Z 122,A 133.1298,B 24.9423,C -1.7551,E1 24.8824,E2 312.9286} C_DIS
LIN {X -84.136,Y 80.3199,Z 122,A 131.633,B 24.9409,C -1.775,E1 24.8852,E2 314.3844} C_DIS
LIN {X -81.7063,Y 82.7884,Z 122,A 130.0155,B 24.9404,C -1.7828,E1 24.8884,E2 315.9901} C_DIS
LIN {X -78.1467,Y 86.1586,Z 122,A 127.0537,B 24.9415,C -1.7662,E1 24.8946,E2 319.0037} C_DIS
LIN {X -75.2363,Y 88.7097,Z 122,A 125.5568,B 24.9401,C -1.7872,E1 24.8976,E2 320.4563} C_DIS
LIN {X -71.805,Y 91.5098,Z 122,A 123.1028,B 24.9406,C -1.7808,E1 24.903,E2 322.9347} C_DIS
LIN {X -69.1802,Y 93.5107,Z 122,A 121.0704,B 24.9414,C -1.7676,E1 24.9077,E2 325.0057} C_DIS
LIN {X -65.1269,Y 96.376,Z 122,A 119.7905,B 24.9379,C -1.8205,E1 24.9104,E2 326.1641} C_DIS
LIN {X -62.8889,Y 97.851,Z 122,A 117.2366,B 24.9411,C -1.7721,E1 24.9167,E2 328.8413} C_DIS
LIN {X -58.3641,Y 100.6166,Z 122,A 115.319,B 24.9389,C -1.8054,E1 24.9211,E2 330.6854} C_DIS
LIN {X -54.8329,Y 102.5851,Z 122,A 113.3652,B 24.9386,C -1.8104,E1 24.9259,E2 332.6329} C_DIS
LIN {X -51.8016,Y 104.1463,Z 122,A 111.7553,B 24.9382,C -1.8161,E1 24.9298,E2 334.2336} C_DIS
LIN {X -48.9376,Y 105.5224,Z 122,A 110.152,B 24.9382,C -1.817,E1 24.9339,E2 335.8389} C_DIS
LIN {X -45.358,Y 107.1099,Z 122,A 108.2437,B 24.9379,C -1.8207,E1 24.9388,E2 337.7428} C_DIS
LIN {X -42.3795,Y 108.3228,Z 122,A 106.8159,B 24.9373,C -1.8295,E1 24.9424,E2 339.153} C_DIS
LIN {X -39.0764,Y 109.5592,Z 122,A 104.7944,B 24.9379,C -1.8198,E1 24.9478,E2 341.2017} C_DIS
LIN {X -35.2652,Y 110.8446,Z 122,A 102.1125,B 24.9398,C -1.7928,E1 24.9551,E2 343.9524} C_DIS
LIN {X -30.2976,Y 112.3027,Z 122,A 100.7472,B 24.9362,C -1.8454,E1 24.9585,E2 345.1949} C_DIS
LIN {X -26.1563,Y 113.3388,Z 122,A 97.8915,B 24.9382,C -1.8155,E1 24.9664,E2 348.1257} C_DIS
LIN {X -22.8854,Y 114.0454,Z 122,A 96.6545,B 24.9369,C -1.8343,E1 24.9697,E2 349.3194} C_DIS
LIN {X -18.1279,Y 114.8971,Z 122,A 93.4573,B 24.9392,C -1.8014,E1 24.9787,E2 352.5978} C_DIS
LIN {X -13.1191,Y 115.5764,Z 122,A 91.6793,B 24.937,C -1.8331,E1 24.9834,E2 354.3018} C_DIS
LIN {X -9.6751,Y 115.9155,Z 122,A 89.9793,B 24.937,C -1.8341,E1 24.9881,E2 356.0001} C_DIS
LIN {X -6.5764,Y 116.1319,Z 122,A 88.4741,B 24.9368,C -1.8358,E1 24.9923,E2 357.5018} C_DIS
LIN {X -3.0072,Y 116.2803,Z 122,A 86.7684,B 24.9366,C -1.8387,E1 24.9971,E2 359.201} C_DIS
LIN {X 0.6427,Y 116.3161,Z 122,A 84.8699,B 24.9369,C -1.8347,E1 25.0024,E2 361.1089} C_DIS
LIN {X 4.5971,Y 116.2276,Z 122,A 82.9946,B 24.9367,C -1.8381,E1 25.0076,E2 362.9759} C_DIS
LIN {X 8.0278,Y 116.0406,Z 122,A 81.4339,B 24.9363,C -1.8438,E1 25.0119,E2 364.5223} C_DIS
LIN {X 12.6384,Y 115.6304,Z 122,A 78.8736,B 24.9371,C -1.8313,E1 25.0191,E2 367.1107} C_DIS
LIN {X 16.1741,Y 115.188,Z 122,A 77.195,B 24.9369,C -1.8342,E1 25.0237,E2 368.7809} C_DIS
LIN {X 21.0428,Y 114.3995,Z 122,A 74.2938,B 24.9384,C -1.8127,E1 25.0319,E2 371.73} C_DIS
LIN {X 24.9403,Y 113.6127,Z 122,A 72.8533,B 24.9369,C -1.8345,E1 25.0356,E2 373.1171} C_DIS
LIN {X 29.0502,Y 112.6319,Z 122,A 70.6445,B 24.9374,C -1.8276,E1 25.0417,E2 375.3389} C_DIS
LIN {X 31.8366,Y 111.8762,Z 122,A 69.002,B 24.9381,C -1.8169,E1 25.0461,E2 377.004} C_DIS
LIN {X 35.1256,Y 110.8897,Z 122,A 67.5918,B 24.9374,C -1.828,E1 25.0498,E2 378.3855} C_DIS
LIN {X 38.1616,Y 109.8802,Z 122,A 66.0666,B 24.9374,C -1.8289,E1 25.0538,E2 379.9055} C_DIS
LIN {X 41.4309,Y 108.6894,Z 122,A 64.3951,B 24.9373,C -1.8292,E1 25.0582,E2 381.5728} C_DIS
LIN {X 44.9066,Y 107.3001,Z 122,A 62.5908,B 24.9373,C -1.829,E1 25.0629,E2 383.3734} C_DIS
LIN {X 48.6359,Y 105.6628,Z 122,A 60.536,B 24.9376,C -1.8245,E1 25.0681,E2 385.4338} C_DIS
LIN {X 51.8827,Y 104.1061,Z 122,A 58.7089,B 24.9379,C -1.8199,E1 25.0727,E2 387.267} C_DIS
LIN {X 55.8665,Y 102.0244,Z 122,A 55.8562,B 24.9401,C -1.7883,E1 25.0799,E2 390.1862} C_DIS
LIN {X 60.0936,Y 99.5928,Z 122,A 54.165,B 24.9381,C -1.8166,E1 25.0838,E2 391.8053} C_DIS
LIN {X 62.6151,Y 98.0268,Z 122,A 52.7577,B 24.9381,C -1.8168,E1 25.0871,E2 393.2076} C_DIS
LIN {X 64.7945,Y 96.6011,Z 122,A 51.2475,B 24.939,C -1.8043,E1 25.0906,E2 394.7421} C_DIS
LIN {X 68.5203,Y 93.9939,Z 122,A 49.466,B 24.9378,C -1.8213,E1 25.0946,E2 396.4773} C_DIS
LIN {X 71.6572,Y 91.6243,Z 122,A 46.7972,B 24.9403,C -1.7845,E1 25.1007,E2 399.2233} C_DIS
LIN {X 74.7107,Y 89.1536,Z 122,A 45.2733,B 24.9393,C -1.7994,E1 25.1039,E2 400.7062} C_DIS
LIN {X 77.9277,Y 86.3558,Z 122,A 43.0759,B 24.9399,C -1.7908,E1 25.1085,E2 402.9152} C_DIS
LIN {X 80.951,Y 83.5277,Z 122,A 41.1412,B 24.9399,C -1.7913,E1 25.1124,E2 404.8408} C_DIS
LIN {X 83.6383,Y 80.8362,Z 122,A 38.7739,B 24.9416,C -1.7646,E1 25.1171,E2 407.261} C_DIS
LIN {X 86.6004,Y 77.6544,Z 122,A 37.2228,B 24.9402,C -1.7867,E1 25.1199,E2 408.7529} C_DIS
LIN {X 89.1589,Y 74.7044,Z 122,A 35.141,B 24.941,C -1.7749,E1 25.1237,E2 410.8531} C_DIS
LIN {X 92.0296,Y 71.1367,Z 122,A 33.1216,B 24.9406,C -1.7804,E1 25.1271,E2 412.8502} C_DIS
LIN {X 93.9652,Y 68.5595,Z 122,A 31.6775,B 24.9404,C -1.7831,E1 25.1295,E2 414.281} C_DIS
LIN {X 97.3066,Y 63.729,Z 122,A 28.52,B 24.9417,C -1.7633,E1 25.1346,E2 417.4696} C_DIS
LIN {X 99.4154,Y 60.3856,Z 122,A 26.6728,B 24.9417,C -1.7628,E1 25.1372,E2 419.3086} C_DIS
LIN {X 101.4819,Y 56.8444,Z 122,A 24.7093,B 24.942,C -1.7599,E1 25.14,E2 421.2688} C_DIS
LIN {X 102.8049,Y 54.4156,Z 122,A 23.0954,B 24.943,C -1.7443,E1 25.1421,E2 422.9108} C_DIS
LIN {X 105.244,Y 49.5357,Z 122,A 20.4707,B 24.9433,C -1.7396,E1 25.1453,E2 425.5325} C_DIS
LIN {X 107.0949,Y 45.3936,Z 122,A 18.4844,B 24.9429,C -1.7448,E1 25.1475,E2 427.4959} C_DIS
LIN {X 108.2632,Y 42.5314,Z 122,A 16.9032,B 24.9434,C -1.7375,E1 25.1492,E2 429.0854} C_DIS
LIN {X 109.6381,Y 38.8516,Z 122,A 14.9781,B 24.9438,C -1.7322,E1 25.151,E2 431.0123} C_DIS
LIN {X 111.3886,Y 33.5053,Z 122,A 11.9881,B 24.945,C -1.7135,E1 25.1536,E2 434.0295} C_DIS
LIN {X 112.943,Y 27.817,Z 122,A 9.358,B 24.9447,C -1.7174,E1 25.1554,E2 436.6352} C_DIS
LIN {X 113.6411,Y 24.8099,Z 122,A 6.7289,B 24.9483,C -1.6608,E1 25.1571,E2 439.3823} C_DIS
LIN {X 114.8883,Y 18.1851,Z 122,A 4.5034,B 24.9458,C -1.7014,E1 25.158,E2 441.4992} C_DIS
LIN {X 115.3526,Y 14.9538,Z 122,A 2.9905,B 24.9458,C -1.7008,E1 25.1586,E2 443.0046} C_DIS
LIN {X 115.7388,Y 11.6029,Z 122,A 1.196,B 24.9465,C -1.6891,E1 25.1591,E2 444.816} C_DIS
LIN {X 116.0552,Y 7.8113,Z 122,A -0.5497,B 24.9465,C -1.6891,E1 25.1595,E2 446.5513} C_DIS
LIN {X 116.2461,Y 4.1204,Z 122,A -2.476,B 24.9472,C -1.6782,E1 25.1597,E2 448.492} C_DIS
LIN {X 116.3181,Y 0.386,Z 122,A -4.3245,B 24.9476,C -1.6718,E1 25.1597,E2 450.3446} C_DIS
LIN {X 116.2651,Y -3.5012,Z 122,A -6.1338,B 24.9477,C -1.6706,E1 25.1597,E2 452.146} C_DIS
LIN {X 116.0908,Y -7.285,Z 122,A -7.9825,B 24.948,C -1.6652,E1 25.1594,E2 453.9962} C_DIS
LIN {X 115.8294,Y -10.6489,Z 122,A -9.6,B 24.9482,C -1.6619,E1 25.159,E2 455.612} C_DIS
LIN {X 115.5589,Y -13.268,Z 122,A -11.8294,B 24.9512,C -1.6138,E1 25.1583,E2 457.9416} C_DIS
LIN {X 114.7353,Y -19.1218,Z 122,A -13.7378,B 24.9489,C -1.6515,E1 25.1575,E2 459.7499} C_DIS
LIN {X 114.159,Y -22.3081,Z 122,A -16.0868,B 24.9514,C -1.6108,E1 25.1562,E2 462.1813} C_DIS
LIN {X 113.1058,Y -27.1494,Z 122,A -17.6087,B 24.9492,C -1.6462,E1 25.1553,E2 463.6107} C_DIS
LIN {X 112.3785,Y -30.0168,Z 122,A -19.5582,B 24.9509,C -1.6182,E1 25.1538,E2 465.6151} C_DIS
LIN {X 110.8692,Y -35.1891,Z 122,A -23.0288,B 24.9537,C -1.5715,E1 25.1509,E2 469.1759} C_DIS
LIN {X 108.5962,Y -41.677,Z 122,A -25.3396,B 24.9514,C -1.6113,E1 25.1487,E2 471.3802} C_DIS
LIN {X 107.2807,Y -44.9526,Z 122,A -26.8811,B 24.9511,C -1.6152,E1 25.1471,E2 472.9039} C_DIS
LIN {X 106.1587,Y -47.542,Z 122,A -28.8906,B 24.9531,C -1.5817,E1 25.1447,E2 474.9813} C_DIS
LIN {X 104.3894,Y -51.3113,Z 122,A -30.4244,B 24.952,C -1.5998,E1 25.1429,E2 476.4643} C_DIS
LIN {X 101.7691,Y -56.3301,Z 122,A -33.2291,B 24.9526,C -1.5908,E1 25.1392,E2 479.2755} C_DIS
LIN {X 100.3221,Y -58.8681,Z 122,A -35.1863,B 24.9543,C -1.5622,E1 25.1364,E2 481.29} C_DIS
LIN {X 98.0318,Y -62.6074,Z 122,A -36.7468,B 24.953,C -1.5841,E1 25.1342,E2 482.791} C_DIS
LIN {X 96.1541,Y -65.4546,Z 122,A -38.3383,B 24.953,C -1.5835,E1 25.1317,E2 484.3761} C_DIS
LIN {X 94.015,Y -68.4916,Z 122,A -40.2385,B 24.9535,C -1.5751,E1 25.1286,E2 486.2868} C_DIS
LIN {X 92.0387,Y -71.1249,Z 122,A -41.8773,B 24.9538,C -1.5699,E1 25.1258,E2 487.9301} C_DIS
LIN {X 89.6055,Y -74.167,Z 122,A -43.7546,B 24.954,C -1.5667,E1 25.1225,E2 489.8063} C_DIS
LIN {X 87.2728,Y -76.8996,Z 122,A -45.6032,B 24.9545,C -1.5583,E1 25.1191,E2 491.6663} C_DIS
LIN {X 84.7149,Y -79.707,Z 122,A -47.3437,B 24.9545,C -1.5597,E1 25.1158,E2 493.3959} C_DIS
LIN {X 82.2507,Y -82.2507,Z 122,A -49.2164,B 24.955,C -1.5493,E1 25.1121,E2 495.285} C_DIS
LIN {X 79.6388,Y -84.7792,Z 122,A -50.8638,B 24.9549,C -1.5517,E1 25.1088,E2 496.92} C_DIS
LIN {X 76.8543,Y -87.3124,Z 122,A -52.7392,B 24.9552,C -1.5464,E1 25.1049,E2 498.8005} C_DIS
LIN {X 74.451,Y -89.3695,Z 122,A -54.252,B 24.9552,C -1.5449,E1 25.1017,E2 500.3109} C_DIS
LIN {X 71.7034,Y -91.5901,Z 122,A -55.9799,B 24.9555,C -1.5416,E1 25.0979,E2 502.0401} C_DIS
LIN {X 68.9753,Y -93.6608,Z 122,A -58.2008,B 24.9571,C -1.5134,E1 25.0928,E2 504.3198} C_DIS
LIN {X 65.668,Y -96.0096,Z 122,A -59.7426,B 24.9561,C -1.5303,E1 25.0894,E2 505.8163} C_DIS
LIN {X 62.5667,Y -98.0579,Z 122,A -61.5139,B 24.9561,C -1.5295,E1 25.0852,E2 507.5839} C_DIS
LIN {X 59.6849,Y -99.8393,Z 122,A -63.3403,B 24.9568,C -1.519,E1 25.0808,E2 509.4291} C_DIS
LIN {X 54.6831,Y -102.664,Z 122,A -66.0366,B 24.9568,C -1.5201,E1 25.0742,E2 512.115} C_DIS
LIN {X 52.173,Y -103.9622,Z 122,A -68.4446,B 24.9594,C -1.4716,E1 25.068,E2 514.6312} C_DIS
LIN {X 46.2895,Y -106.7107,Z 122,A -70.5498,B 24.9569,C -1.5163,E1 25.0629,E2 516.6257} C_DIS
LIN {X 42.7218,Y -108.1884,Z 122,A -72.4656,B 24.9571,C -1.5129,E1 25.0579,E2 518.5451} C_DIS
LIN {X 36.604,Y -110.4082,Z 122,A -75.9977,B 24.9582,C -1.4939,E1 25.0485,E2 522.115} C_DIS
LIN {X 33.4512,Y -111.4047,Z 122,A -77.0687,B 24.9569,C -1.5173,E1 25.0458,E2 523.1287} C_DIS
LIN {X 26.4137,Y -113.2793,Z 122,A -80.5829,B 24.9569,C -1.5167,E1 25.0363,E2 526.6387} C_DIS
LIN {X 21.3732,Y -114.3391,Z 122,A -83.4663,B 24.9579,C -1.4988,E1 25.0283,E2 529.5611} C_DIS
LIN {X 18.0036,Y -114.9163,Z 122,A -85.0861,B 24.9579,C -1.5004,E1 25.0239,E2 531.1754} C_DIS
LIN {X 13.8216,Y -115.4941,Z 122,A -87.1571,B 24.9579,C -1.4994,E1 25.0181,E2 533.247} C_DIS
LIN {X 10.4093,Y -115.8515,Z 122,A -88.9297,B 24.9581,C -1.4948,E1 25.0132,E2 535.0294} C_DIS
LIN {X 6.2873,Y -116.1478,Z 122,A -90.923,B 24.9581,C -1.4958,E1 25.0076,E2 537.0196} C_DIS
LIN {X 2.3788,Y -116.2937,Z 122,A -92.797,B 24.958,C -1.4975,E1 25.0024,E2 538.8891} C_DIS
LIN {X 2.3788,Y -116.2937,Z 122,A -92.797,B 24.958,C -1.4975,E1 25.0024,E2 538.8891} C_DIS
Enddeposition()
LIN {X 0.8123,Y -115.4362,Z 122,A -93.413,B 24.9567,C -1.5197,E1 25.0009,E2 539.4525} C_DIS
Startdeposition()
$VEL.CP = VEL_PRINT
LIN {X 3.4427,Y -115.3894,Z 122,A -91.5404,B 24.9553,C -1.5453,E1 25.0062,E2 537.5196} C_DIS
LIN {X 7.0427,Y -115.2276,Z 122,A -89.6552,B 24.955,C -1.5503,E1 25.0115,E2 535.6232} C_DIS
LIN {X 10.6634,Y -114.9472,Z 122,A -87.9696,B 24.9552,C -1.546,E1 25.0162,E2 533.9487} C_DIS
LIN {X 14.0985,Y -114.5786,Z 122,A -86.052,B 24.9546,C -1.5562,E1 25.0216,E2 532.0084} C_DIS
LIN {X 17.7265,Y -114.0716,Z 122,A -84.4964,B 24.9552,C -1.5456,E1 25.0258,E2 530.4793} C_DIS
LIN {X 20.6153,Y -113.5852,Z 122,A -82.0083,B 24.9524,C -1.594,E1 25.033,E2 527.8794} C_DIS
LIN {X 26.4857,Y -112.3625,Z 122,A -79.9758,B 24.9548,C -1.5535,E1 25.0382,E2 525.9455} C_DIS
LIN {X 32.8,Y -110.683,Z 122,A -76.8008,B 24.9548,C -1.5539,E1 25.0468,E2 522.7746} C_DIS
LIN {X 35.9306,Y -109.7074,Z 122,A -74.3431,B 24.9524,C -1.5941,E1 25.0535,E2 520.2265} C_DIS
LIN {X 40.8283,Y -107.9797,Z 122,A -72.5678,B 24.9544,C -1.5605,E1 25.0579,E2 518.5344} C_DIS
LIN {X 43.9924,Y -106.7309,Z 122,A -70.7724,B 24.9539,C -1.5679,E1 25.0626,E2 516.7258} C_DIS
LIN {X 50.3976,Y -103.8597,Z 122,A -67.6217,B 24.9545,C -1.5579,E1 25.0705,E2 513.6064} C_DIS
Enddeposition()
END
